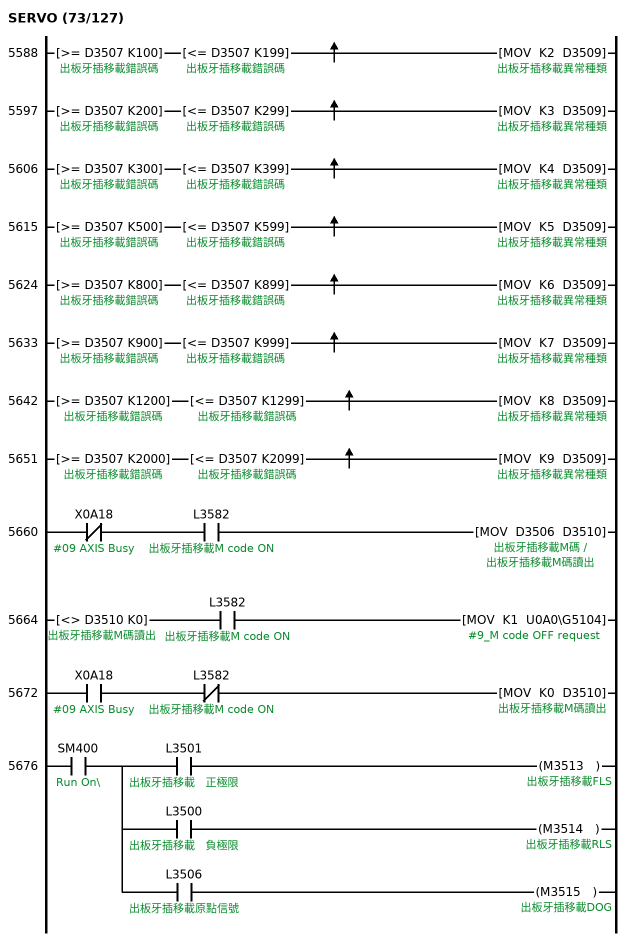
[picture p72: ladder of SERVO, rungs at steps 5588 to 5676]
5588  LD>=    D3507 K100  ; 出板牙插移載錯誤碼
      AND<=   D3507 K199  ; 出板牙插移載錯誤碼
      MEP
      MOV     K2 D3509
5597  LD>=    D3507 K200  ; 出板牙插移載錯誤碼
      AND<=   D3507 K299  ; 出板牙插移載錯誤碼
      MEP
      MOV     K3 D3509
5606  LD>=    D3507 K300  ; 出板牙插移載錯誤碼
      AND<=   D3507 K399  ; 出板牙插移載錯誤碼
      MEP
      MOV     K4 D3509
5615  LD>=    D3507 K500  ; 出板牙插移載錯誤碼
      AND<=   D3507 K599  ; 出板牙插移載錯誤碼
      MEP
      MOV     K5 D3509
5624  LD>=    D3507 K800  ; 出板牙插移載錯誤碼
      AND<=   D3507 K899  ; 出板牙插移載錯誤碼
      MEP
      MOV     K6 D3509
5633  LD>=    D3507 K900  ; 出板牙插移載錯誤碼
      AND<=   D3507 K999  ; 出板牙插移載錯誤碼
      MEP
      MOV     K7 D3509
5642  LD>=    D3507 K1200  ; 出板牙插移載錯誤碼
      AND<=   D3507 K1299  ; 出板牙插移載錯誤碼
      MEP
      MOV     K8 D3509
5651  LD>=    D3507 K2000  ; 出板牙插移載錯誤碼
      AND<=   D3507 K2099  ; 出板牙插移載錯誤碼
      MEP
      MOV     K9 D3509
5660  LDI     X0A18  ; #09 AXIS Busy
      AND     L3582  ; 出板牙插移載M code ON
      MOV     D3506 D3510  ; 出板牙插移載M碼讀出
5664  LD<>    D3510 K0  ; 出板牙插移載M碼讀出
      AND     L3582  ; 出板牙插移載M code ON
      MOV     K1 U0A0\G5104  ; #9_M code OFF request
5672  LD      X0A18  ; #09 AXIS Busy
      ANI     L3582  ; 出板牙插移載M code ON
      MOV     K0 D3510
5676  LD      SM400  ; Run On\
      MPS
      AND     L3501  ; 出板牙插移載   正極限
      OUT     M3513  ; 出板牙插移載FLS
      MRD
      AND     L3500  ; 出板牙插移載   負極限
      OUT     M3514  ; 出板牙插移載RLS
      MPP
      AND     L3506  ; 出板牙插移載原點信號
      OUT     M3515  ; 出板牙插移載DOG
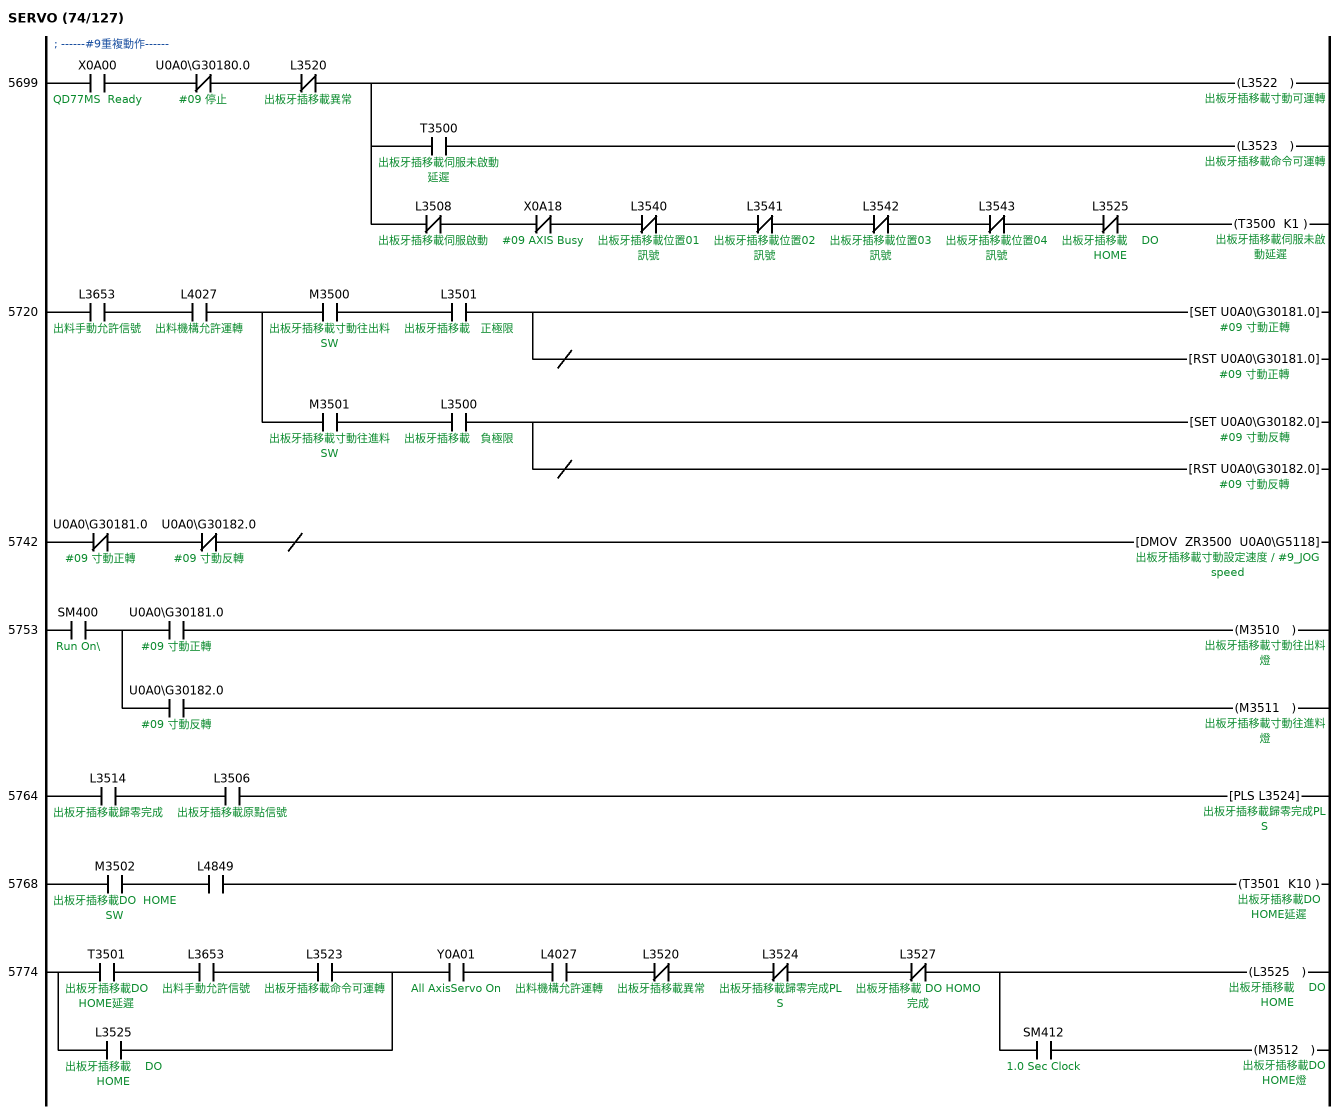
; ------#9重複動作------
5699  LD      X0A00  ; QD77MS  Ready
      ANI     U0A0\G30180.0  ; #09 停止
      ANI     L3520  ; 出板牙插移載異常
      OUT     L3522  ; 出板牙插移載寸動可運轉
      MPS
      AND     T3500  ; 出板牙插移載伺服未啟動延遲
      OUT     L3523  ; 出板牙插移載命令可運轉
      MPP
      ANI     L3508  ; 出板牙插移載伺服啟動
      ANI     X0A18  ; #09 AXIS Busy
      ANI     L3540  ; 出板牙插移載位置01 訊號
      ANI     L3541  ; 出板牙插移載位置02 訊號
      ANI     L3542  ; 出板牙插移載位置03 訊號
      ANI     L3543  ; 出板牙插移載位置04 訊號
      ANI     L3525  ; 出板牙插移載    DO HOME
      OUT     T3500 K1  ; 出板牙插移載伺服未啟動延遲
5720  LD      L3653  ; 出料手動允許信號
      AND     L4027  ; 出料機構允許運轉
      MPS
      AND     M3500  ; 出板牙插移載寸動往出料SW
      AND     L3501  ; 出板牙插移載   正極限
      SET     U0A0\G30181.0  ; #09 寸動正轉
      INV
      RST     U0A0\G30181.0  ; #09 寸動正轉
      MPP
      AND     M3501  ; 出板牙插移載寸動往進料SW
      AND     L3500  ; 出板牙插移載   負極限
      SET     U0A0\G30182.0  ; #09 寸動反轉
      INV
      RST     U0A0\G30182.0  ; #09 寸動反轉
5742  LDI     U0A0\G30181.0  ; #09 寸動正轉
      ANI     U0A0\G30182.0  ; #09 寸動反轉
      INV
      DMOV    ZR3500 U0A0\G5118  ; 出板牙插移載寸動設定速度 / #9_JOG     speed
5753  LD      SM400  ; Run On\
      MPS
      AND     U0A0\G30181.0  ; #09 寸動正轉
      OUT     M3510  ; 出板牙插移載寸動往出料燈
      MPP
      AND     U0A0\G30182.0  ; #09 寸動反轉
      OUT     M3511  ; 出板牙插移載寸動往進料燈
5764  LD      L3514  ; 出板牙插移載歸零完成
      AND     L3506  ; 出板牙插移載原點信號
      PLS     L3524  ; 出板牙插移載歸零完成PLS
5768  LD      M3502  ; 出板牙插移載DO  HOME SW
      AND     L4849
      OUT     T3501 K10  ; 出板牙插移載DO HOME延遲
5774  LD      T3501  ; 出板牙插移載DO HOME延遲
      AND     L3653  ; 出料手動允許信號
      AND     L3523  ; 出板牙插移載命令可運轉
      OR      L3525  ; 出板牙插移載    DO HOME
      AND     Y0A01  ; All AxisServo On
      AND     L4027  ; 出料機構允許運轉
      ANI     L3520  ; 出板牙插移載異常
      ANI     L3524  ; 出板牙插移載歸零完成PLS
      ANI     L3527  ; 出板牙插移載 DO HOMO 完成
      OUT     L3525  ; 出板牙插移載    DO HOME
      AND     SM412  ; 1.0 Sec Clock
      OUT     M3512  ; 出板牙插移載DO  HOME燈
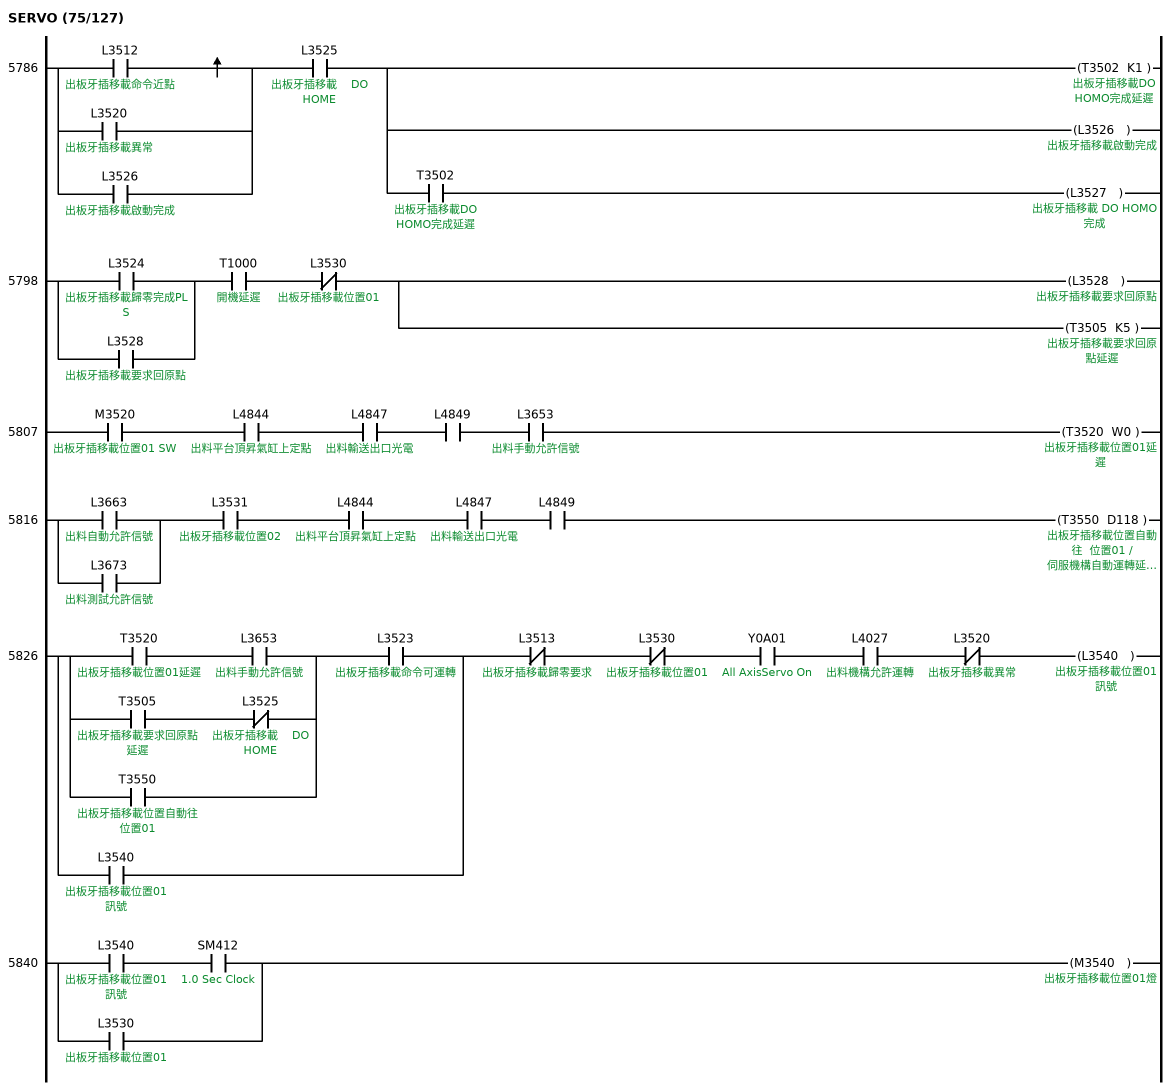
5786  LD      L3512  ; 出板牙插移載命令近點
      MEP
      OR      L3520  ; 出板牙插移載異常
      OR      L3526  ; 出板牙插移載啟動完成
      AND     L3525  ; 出板牙插移載    DO HOME
      OUT     T3502 K1  ; 出板牙插移載DO HOMO完成延遲
      OUT     L3526  ; 出板牙插移載啟動完成
      AND     T3502  ; 出板牙插移載DO HOMO完成延遲
      OUT     L3527  ; 出板牙插移載 DO HOMO 完成
5798  LD      L3524  ; 出板牙插移載歸零完成PLS
      OR      L3528  ; 出板牙插移載要求回原點
      AND     T1000  ; 開機延遲
      ANI     L3530  ; 出板牙插移載位置01
      OUT     L3528  ; 出板牙插移載要求回原點
      OUT     T3505 K5  ; 出板牙插移載要求回原點延遲
5807  LD      M3520  ; 出板牙插移載位置01 SW
      AND     L4844  ; 出料平台頂昇氣缸上定點
      AND     L4847  ; 出料輸送出口光電
      AND     L4849
      AND     L3653  ; 出料手動允許信號
      OUT     T3520 W0  ; 出板牙插移載位置01延遲
5816  LD      L3663  ; 出料自動允許信號
      OR      L3673  ; 出料測試允許信號
      AND     L3531  ; 出板牙插移載位置02
      AND     L4844  ; 出料平台頂昇氣缸上定點
      AND     L4847  ; 出料輸送出口光電
      AND     L4849
      OUT     T3550 D118  ; 出板牙插移載位置自動往  位置01 / 伺服機構自動運轉延遲時間
5826  LD      T3520  ; 出板牙插移載位置01延遲
      AND     L3653  ; 出料手動允許信號
      LD      T3505  ; 出板牙插移載要求回原點延遲
      ANI     L3525  ; 出板牙插移載    DO HOME
      ORB
      OR      T3550  ; 出板牙插移載位置自動往  位置01
      AND     L3523  ; 出板牙插移載命令可運轉
      OR      L3540  ; 出板牙插移載位置01 訊號
      ANI     L3513  ; 出板牙插移載歸零要求
      ANI     L3530  ; 出板牙插移載位置01
      AND     Y0A01  ; All AxisServo On
      AND     L4027  ; 出料機構允許運轉
      ANI     L3520  ; 出板牙插移載異常
      OUT     L3540  ; 出板牙插移載位置01 訊號
5840  LD      L3540  ; 出板牙插移載位置01 訊號
      AND     SM412  ; 1.0 Sec Clock
      OR      L3530  ; 出板牙插移載位置01
      OUT     M3540  ; 出板牙插移載位置01燈
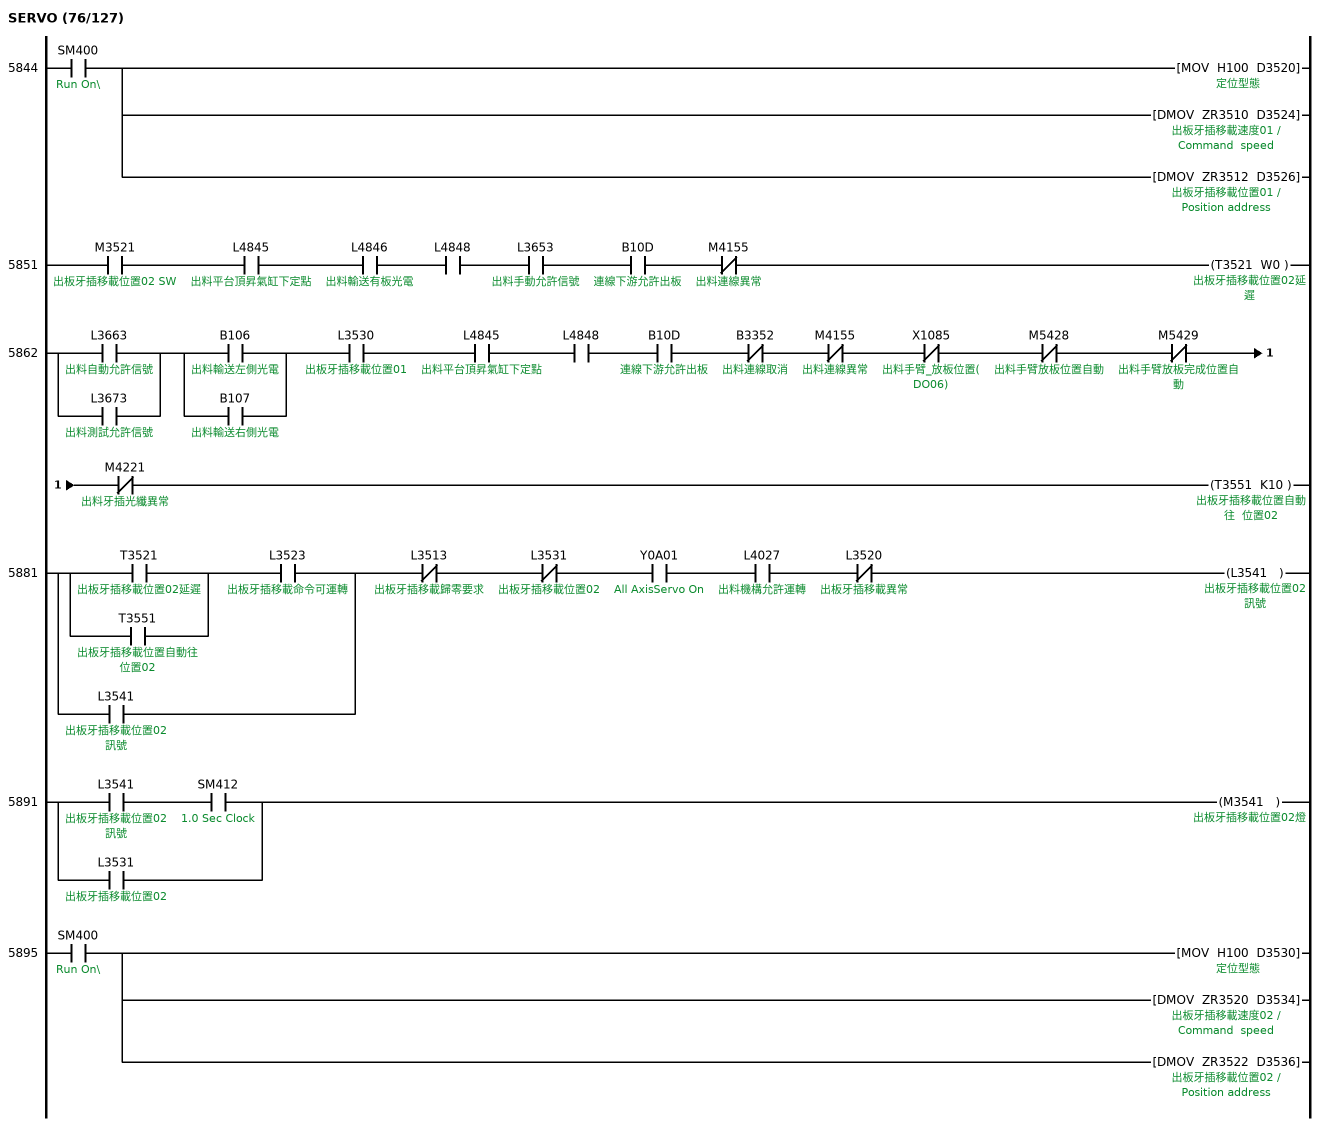
5844  LD      SM400  ; Run On\
      MOV     H100 D3520  ; 定位型態
      DMOV    ZR3510 D3524  ; 出板牙插移載速度01 / Command  speed
      DMOV    ZR3512 D3526  ; Position address
5851  LD      M3521  ; 出板牙插移載位置02 SW
      AND     L4845  ; 出料平台頂昇氣缸下定點
      AND     L4846  ; 出料輸送有板光電
      AND     L4848
      AND     L3653  ; 出料手動允許信號
      AND     B10D  ; 連線下游允許出板
      ANI     M4155  ; 出料連線異常
      OUT     T3521 W0  ; 出板牙插移載位置02延遲
5862  LD      L3663  ; 出料自動允許信號
      OR      L3673  ; 出料測試允許信號
      LD      B106  ; 出料輸送左側光電
      OR      B107  ; 出料輸送右側光電
      ANB
      AND     L3530  ; 出板牙插移載位置01
      AND     L4845  ; 出料平台頂昇氣缸下定點
      AND     L4848
      AND     B10D  ; 連線下游允許出板
      ANI     B3352  ; 出料連線取消
      ANI     M4155  ; 出料連線異常
      ANI     X1085  ; 出料手臂_放板位置(DO06)
      ANI     M5428  ; 出料手臂放板位置自動
      ANI     M5429  ; 出料手臂放板完成位置自動
      ANI     M4221  ; 出料牙插光纖異常
      OUT     T3551 K10  ; 出板牙插移載位置自動往  位置02
5881  LD      T3521  ; 出板牙插移載位置02延遲
      OR      T3551  ; 出板牙插移載位置自動往  位置02
      AND     L3523  ; 出板牙插移載命令可運轉
      OR      L3541  ; 出板牙插移載位置02 訊號
      ANI     L3513  ; 出板牙插移載歸零要求
      ANI     L3531  ; 出板牙插移載位置02
      AND     Y0A01  ; All AxisServo On
      AND     L4027  ; 出料機構允許運轉
      ANI     L3520  ; 出板牙插移載異常
      OUT     L3541  ; 出板牙插移載位置02 訊號
5891  LD      L3541  ; 出板牙插移載位置02 訊號
      AND     SM412  ; 1.0 Sec Clock
      OR      L3531  ; 出板牙插移載位置02
      OUT     M3541  ; 出板牙插移載位置02燈
5895  LD      SM400  ; Run On\
      MOV     H100 D3530  ; 定位型態
      DMOV    ZR3520 D3534  ; 出板牙插移載速度02 / Command  speed
      DMOV    ZR3522 D3536  ; Position address
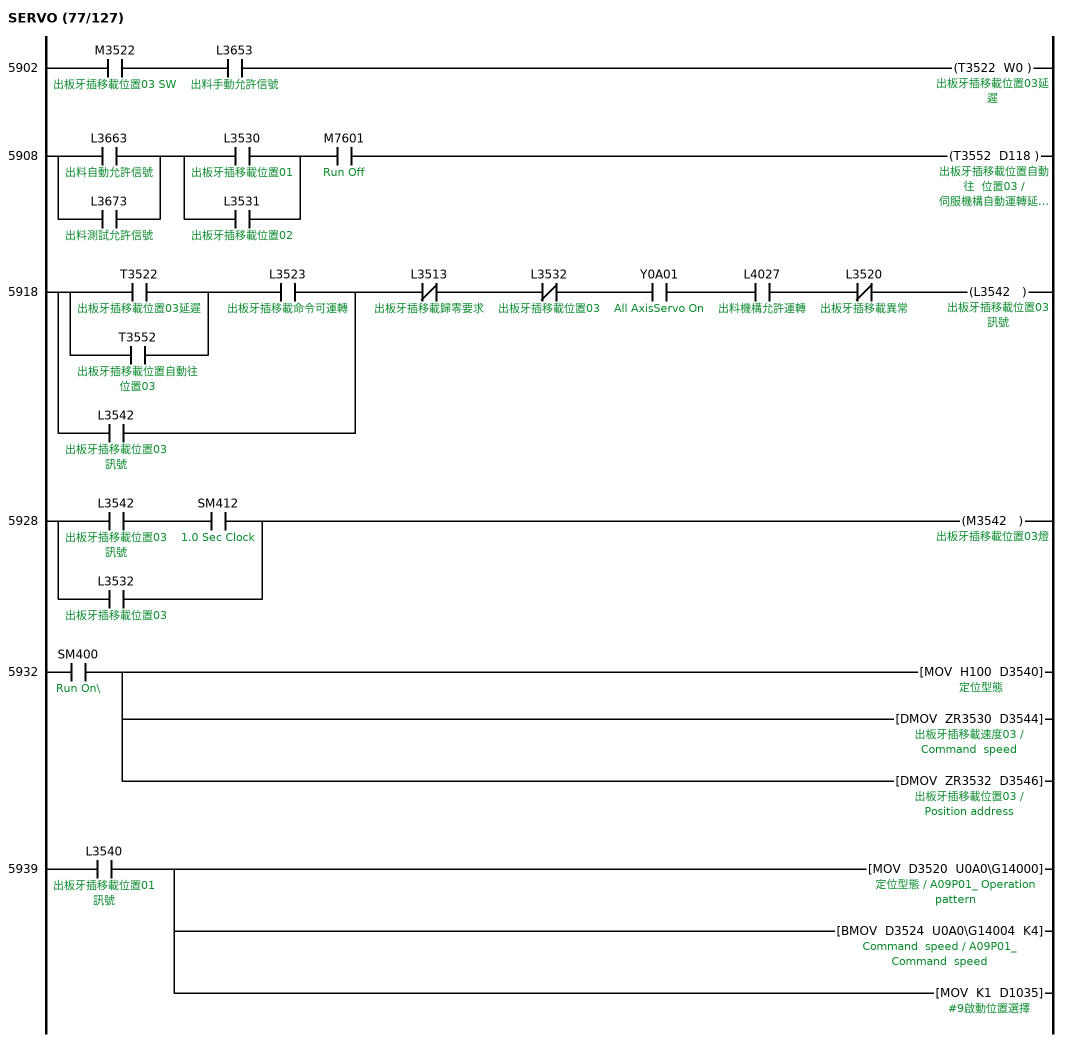
5902  LD      M3522  ; 出板牙插移載位置03 SW
      AND     L3653  ; 出料手動允許信號
      OUT     T3522 W0  ; 出板牙插移載位置03延遲
5908  LD      L3663  ; 出料自動允許信號
      OR      L3673  ; 出料測試允許信號
      LD      L3530  ; 出板牙插移載位置01
      OR      L3531  ; 出板牙插移載位置02
      ANB
      AND     M7601  ; Run Off
      OUT     T3552 D118  ; 出板牙插移載位置自動往  位置03 / 伺服機構自動運轉延遲時間
5918  LD      T3522  ; 出板牙插移載位置03延遲
      OR      T3552  ; 出板牙插移載位置自動往  位置03
      AND     L3523  ; 出板牙插移載命令可運轉
      OR      L3542  ; 出板牙插移載位置03 訊號
      ANI     L3513  ; 出板牙插移載歸零要求
      ANI     L3532  ; 出板牙插移載位置03
      AND     Y0A01  ; All AxisServo On
      AND     L4027  ; 出料機構允許運轉
      ANI     L3520  ; 出板牙插移載異常
      OUT     L3542  ; 出板牙插移載位置03 訊號
5928  LD      L3542  ; 出板牙插移載位置03 訊號
      AND     SM412  ; 1.0 Sec Clock
      OR      L3532  ; 出板牙插移載位置03
      OUT     M3542  ; 出板牙插移載位置03燈
5932  LD      SM400  ; Run On\
      MOV     H100 D3540  ; 定位型態
      DMOV    ZR3530 D3544  ; 出板牙插移載速度03 / Command  speed
      DMOV    ZR3532 D3546  ; Position address
5939  LD      L3540  ; 出板牙插移載位置01 訊號
      MOV     D3520 U0A0\G14000  ; A09P01_ Operation pattern
      BMOV    D3524 U0A0\G14004 K4  ; A09P01_ Command  speed
      MOV     K1 D1035  ; #9啟動位置選擇
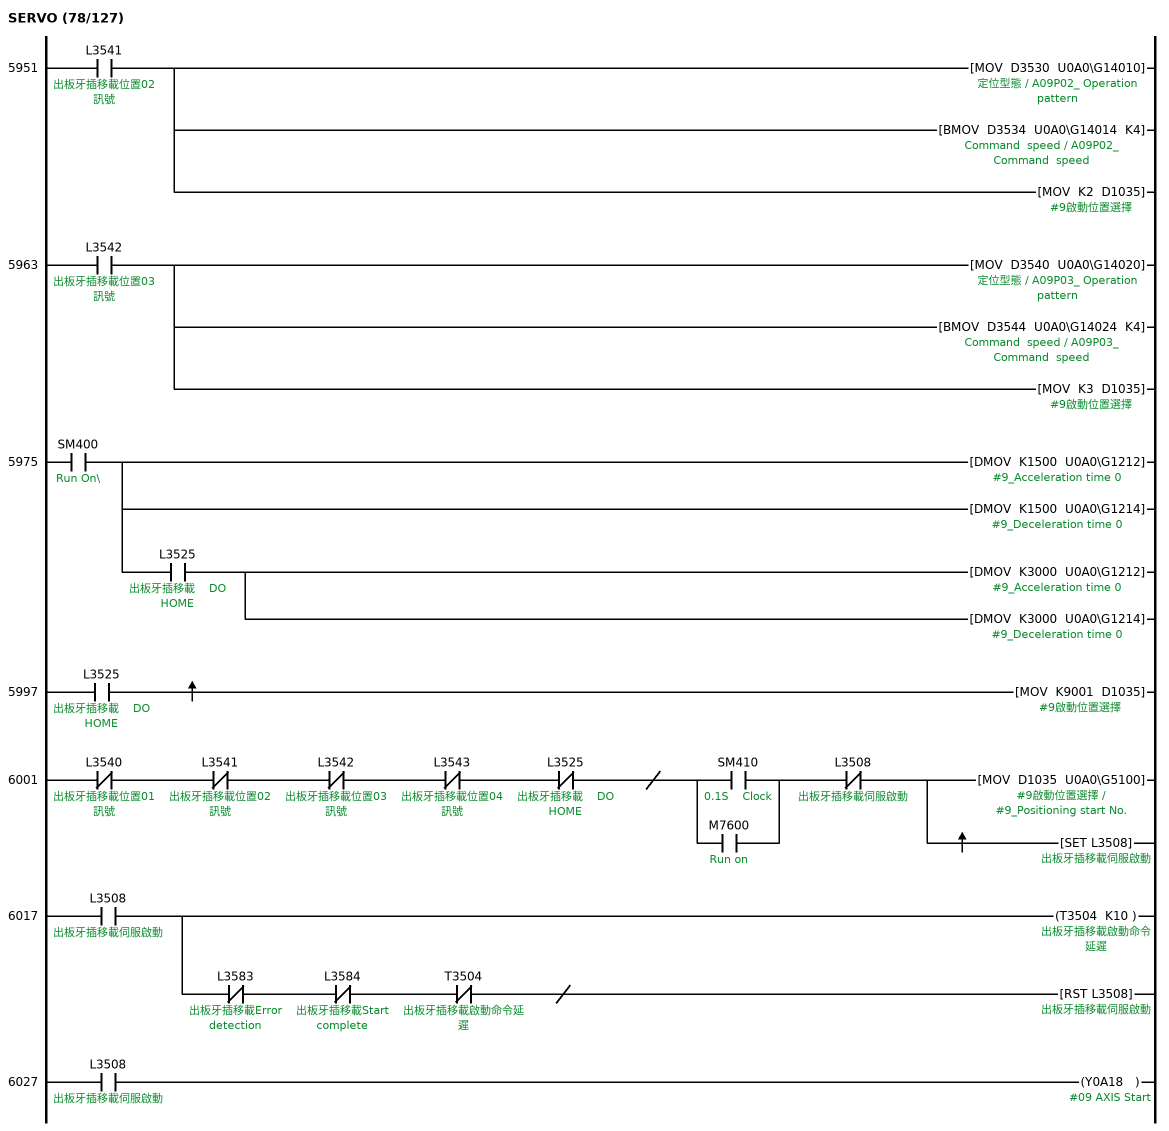
5951  LD      L3541  ; 出板牙插移載位置02 訊號
      MOV     D3530 U0A0\G14010  ; A09P02_ Operation pattern
      BMOV    D3534 U0A0\G14014 K4  ; A09P02_ Command  speed
      MOV     K2 D1035
5963  LD      L3542  ; 出板牙插移載位置03 訊號
      MOV     D3540 U0A0\G14020  ; A09P03_ Operation pattern
      BMOV    D3544 U0A0\G14024 K4  ; A09P03_ Command  speed
      MOV     K3 D1035
5975  LD      SM400  ; Run On\
      DMOV    K1500 U0A0\G1212  ; #9_Acceleration time 0
      DMOV    K1500 U0A0\G1214  ; #9_Deceleration time 0
      AND     L3525  ; 出板牙插移載    DO HOME
      DMOV    K3000 U0A0\G1212
      DMOV    K3000 U0A0\G1214
5997  LD      L3525  ; 出板牙插移載    DO HOME
      MEP
      MOV     K9001 D1035
6001  LDI     L3540  ; 出板牙插移載位置01 訊號
      ANI     L3541  ; 出板牙插移載位置02 訊號
      ANI     L3542  ; 出板牙插移載位置03 訊號
      ANI     L3543  ; 出板牙插移載位置04 訊號
      ANI     L3525  ; 出板牙插移載    DO HOME
      INV
      LD      SM410  ; 0.1S    Clock
      OR      M7600  ; Run on
      ANB
      ANI     L3508  ; 出板牙插移載伺服啟動
      MOV     D1035 U0A0\G5100  ; #9_Positioning start No.
      MEP
      SET     L3508  ; 出板牙插移載伺服啟動
6017  LD      L3508  ; 出板牙插移載伺服啟動
      OUT     T3504 K10  ; 出板牙插移載啟動命令延遲
      ANI     L3583  ; 出板牙插移載Error detection
      ANI     L3584  ; 出板牙插移載Start complete
      ANI     T3504  ; 出板牙插移載啟動命令延遲
      INV
      RST     L3508  ; 出板牙插移載伺服啟動
6027  LD      L3508  ; 出板牙插移載伺服啟動
      OUT     Y0A18  ; #09 AXIS Start
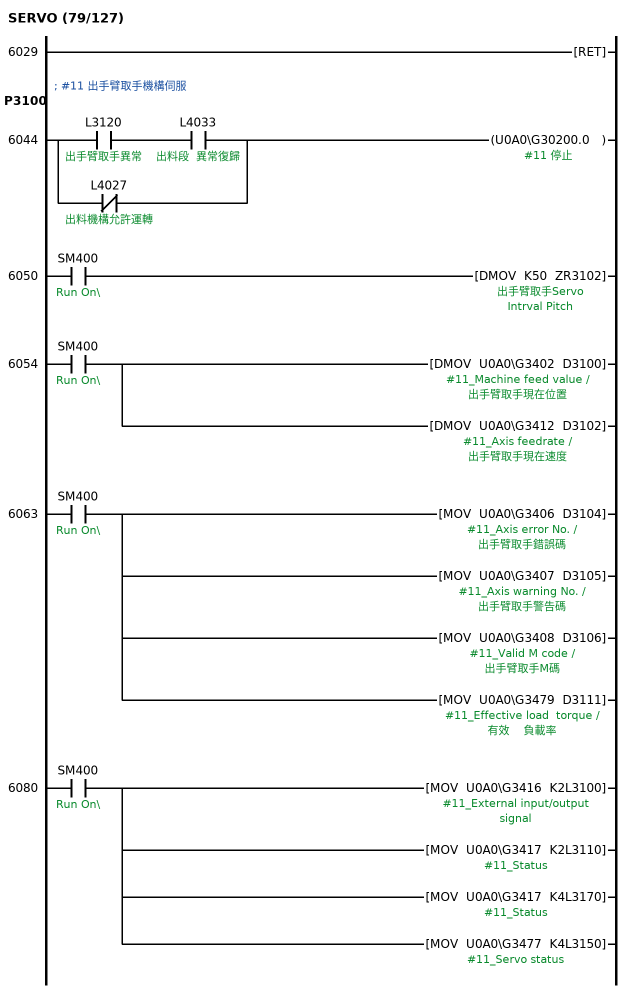
6029  RET
; #11 出手臂取手機構伺服
      P3100
6044  LD      L3120  ; 出手臂取手異常
      AND     L4033  ; 出料段  異常復歸
      ORI     L4027  ; 出料機構允許運轉
      OUT     U0A0\G30200.0  ; #11 停止
6050  LD      SM400  ; Run On\
      DMOV    K50 ZR3102  ; 出手臂取手Servo   Intrval Pitch
6054  LD      SM400  ; Run On\
      DMOV    U0A0\G3402 D3100  ; #11_Machine feed value / 出手臂取手現在位置
      DMOV    U0A0\G3412 D3102  ; #11_Axis feedrate / 出手臂取手現在速度
6063  LD      SM400  ; Run On\
      MOV     U0A0\G3406 D3104  ; #11_Axis error No. / 出手臂取手錯誤碼
      MOV     U0A0\G3407 D3105  ; #11_Axis warning No. / 出手臂取手警告碼
      MOV     U0A0\G3408 D3106  ; #11_Valid M code / 出手臂取手M碼
      MOV     U0A0\G3479 D3111  ; #11_Effective load  torque / 有效    負載率
6080  LD      SM400  ; Run On\
      MOV     U0A0\G3416 K2L3100  ; #11_External input/output signal / 出手臂取手     負極限
      MOV     U0A0\G3417 K2L3110  ; #11_Status / 出手臂取手速度控制
      MOV     U0A0\G3417 K4L3170  ; 出手臂取手速度控制
      MOV     U0A0\G3477 K4L3150  ; #11_Servo status / READY ON
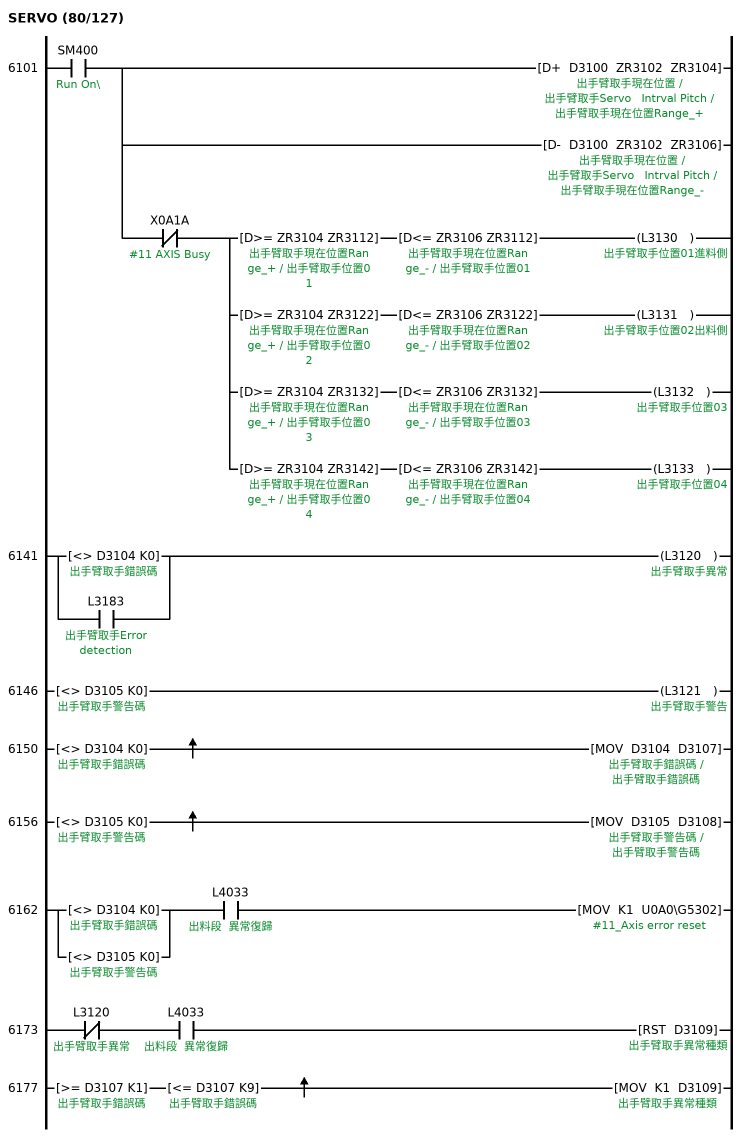
6101  LD      SM400  ; Run On\
      D+      D3100 ZR3102 ZR3104  ; 出手臂取手現在位置Range_+
      D-      D3100 ZR3102 ZR3106  ; 出手臂取手現在位置Range_-
      ANI     X0A1A  ; #11 AXIS Busy
      MPS
      ANDD>=  ZR3104 ZR3112  ; 出手臂取手現在位置Range_+ / 出手臂取手位置01
      ANDD<=  ZR3106 ZR3112  ; 出手臂取手現在位置Range_- / 出手臂取手位置01
      OUT     L3130  ; 出手臂取手位置01進料側
      MRD
      ANDD>=  ZR3104 ZR3122  ; 出手臂取手現在位置Range_+ / 出手臂取手位置02
      ANDD<=  ZR3106 ZR3122  ; 出手臂取手現在位置Range_- / 出手臂取手位置02
      OUT     L3131  ; 出手臂取手位置02出料側
      MRD
      ANDD>=  ZR3104 ZR3132  ; 出手臂取手現在位置Range_+ / 出手臂取手位置03
      ANDD<=  ZR3106 ZR3132  ; 出手臂取手現在位置Range_- / 出手臂取手位置03
      OUT     L3132  ; 出手臂取手位置03
      MPP
      ANDD>=  ZR3104 ZR3142  ; 出手臂取手現在位置Range_+ / 出手臂取手位置04
      ANDD<=  ZR3106 ZR3142  ; 出手臂取手現在位置Range_- / 出手臂取手位置04
      OUT     L3133  ; 出手臂取手位置04
6141  LD<>    D3104 K0  ; 出手臂取手錯誤碼
      OR      L3183  ; 出手臂取手Error detection
      OUT     L3120  ; 出手臂取手異常
6146  LD<>    D3105 K0  ; 出手臂取手警告碼
      OUT     L3121  ; 出手臂取手警告
6150  LD<>    D3104 K0  ; 出手臂取手錯誤碼
      MEP
      MOV     D3104 D3107  ; 出手臂取手錯誤碼
6156  LD<>    D3105 K0  ; 出手臂取手警告碼
      MEP
      MOV     D3105 D3108  ; 出手臂取手警告碼
6162  LD<>    D3104 K0  ; 出手臂取手錯誤碼
      OR<>    D3105 K0  ; 出手臂取手警告碼
      AND     L4033  ; 出料段  異常復歸
      MOV     K1 U0A0\G5302  ; #11_Axis error reset
6173  LDI     L3120  ; 出手臂取手異常
      AND     L4033  ; 出料段  異常復歸
      RST     D3109  ; 出手臂取手異常種類
6177  LD>=    D3107 K1  ; 出手臂取手錯誤碼
      AND<=   D3107 K9  ; 出手臂取手錯誤碼
      MEP
      MOV     K1 D3109
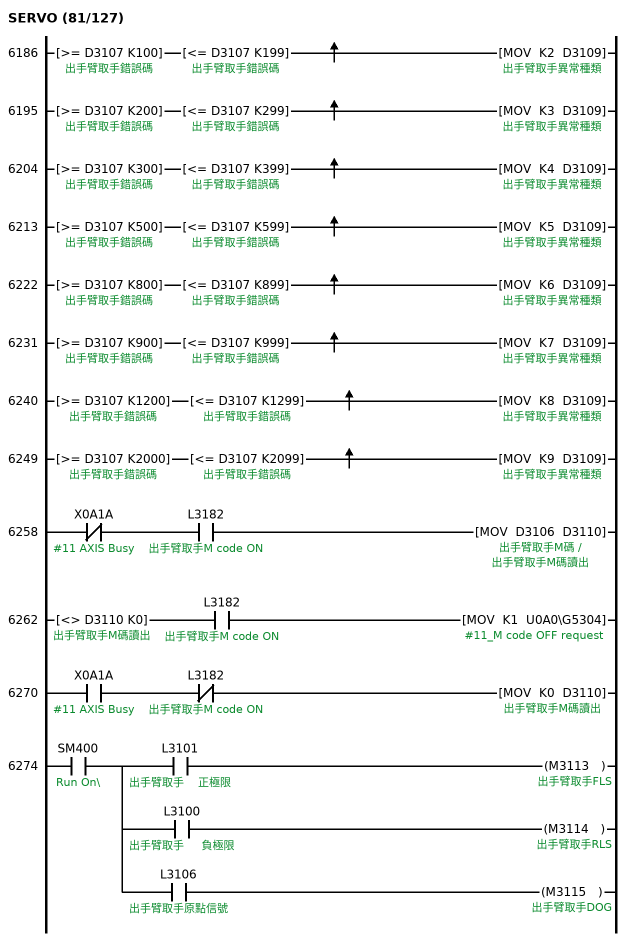
6186  LD>=    D3107 K100  ; 出手臂取手錯誤碼
      AND<=   D3107 K199  ; 出手臂取手錯誤碼
      MEP
      MOV     K2 D3109
6195  LD>=    D3107 K200  ; 出手臂取手錯誤碼
      AND<=   D3107 K299  ; 出手臂取手錯誤碼
      MEP
      MOV     K3 D3109
6204  LD>=    D3107 K300  ; 出手臂取手錯誤碼
      AND<=   D3107 K399  ; 出手臂取手錯誤碼
      MEP
      MOV     K4 D3109
6213  LD>=    D3107 K500  ; 出手臂取手錯誤碼
      AND<=   D3107 K599  ; 出手臂取手錯誤碼
      MEP
      MOV     K5 D3109
6222  LD>=    D3107 K800  ; 出手臂取手錯誤碼
      AND<=   D3107 K899  ; 出手臂取手錯誤碼
      MEP
      MOV     K6 D3109
6231  LD>=    D3107 K900  ; 出手臂取手錯誤碼
      AND<=   D3107 K999  ; 出手臂取手錯誤碼
      MEP
      MOV     K7 D3109
6240  LD>=    D3107 K1200  ; 出手臂取手錯誤碼
      AND<=   D3107 K1299  ; 出手臂取手錯誤碼
      MEP
      MOV     K8 D3109
6249  LD>=    D3107 K2000  ; 出手臂取手錯誤碼
      AND<=   D3107 K2099  ; 出手臂取手錯誤碼
      MEP
      MOV     K9 D3109
6258  LDI     X0A1A  ; #11 AXIS Busy
      AND     L3182  ; 出手臂取手M code ON
      MOV     D3106 D3110  ; 出手臂取手M碼讀出
6262  LD<>    D3110 K0  ; 出手臂取手M碼讀出
      AND     L3182  ; 出手臂取手M code ON
      MOV     K1 U0A0\G5304  ; #11_M code OFF request
6270  LD      X0A1A  ; #11 AXIS Busy
      ANI     L3182  ; 出手臂取手M code ON
      MOV     K0 D3110
6274  LD      SM400  ; Run On\
      MPS
      AND     L3101  ; 出手臂取手    正極限
      OUT     M3113  ; 出手臂取手FLS
      MRD
      AND     L3100  ; 出手臂取手     負極限
      OUT     M3114  ; 出手臂取手RLS
      MPP
      AND     L3106  ; 出手臂取手原點信號
      OUT     M3115  ; 出手臂取手DOG
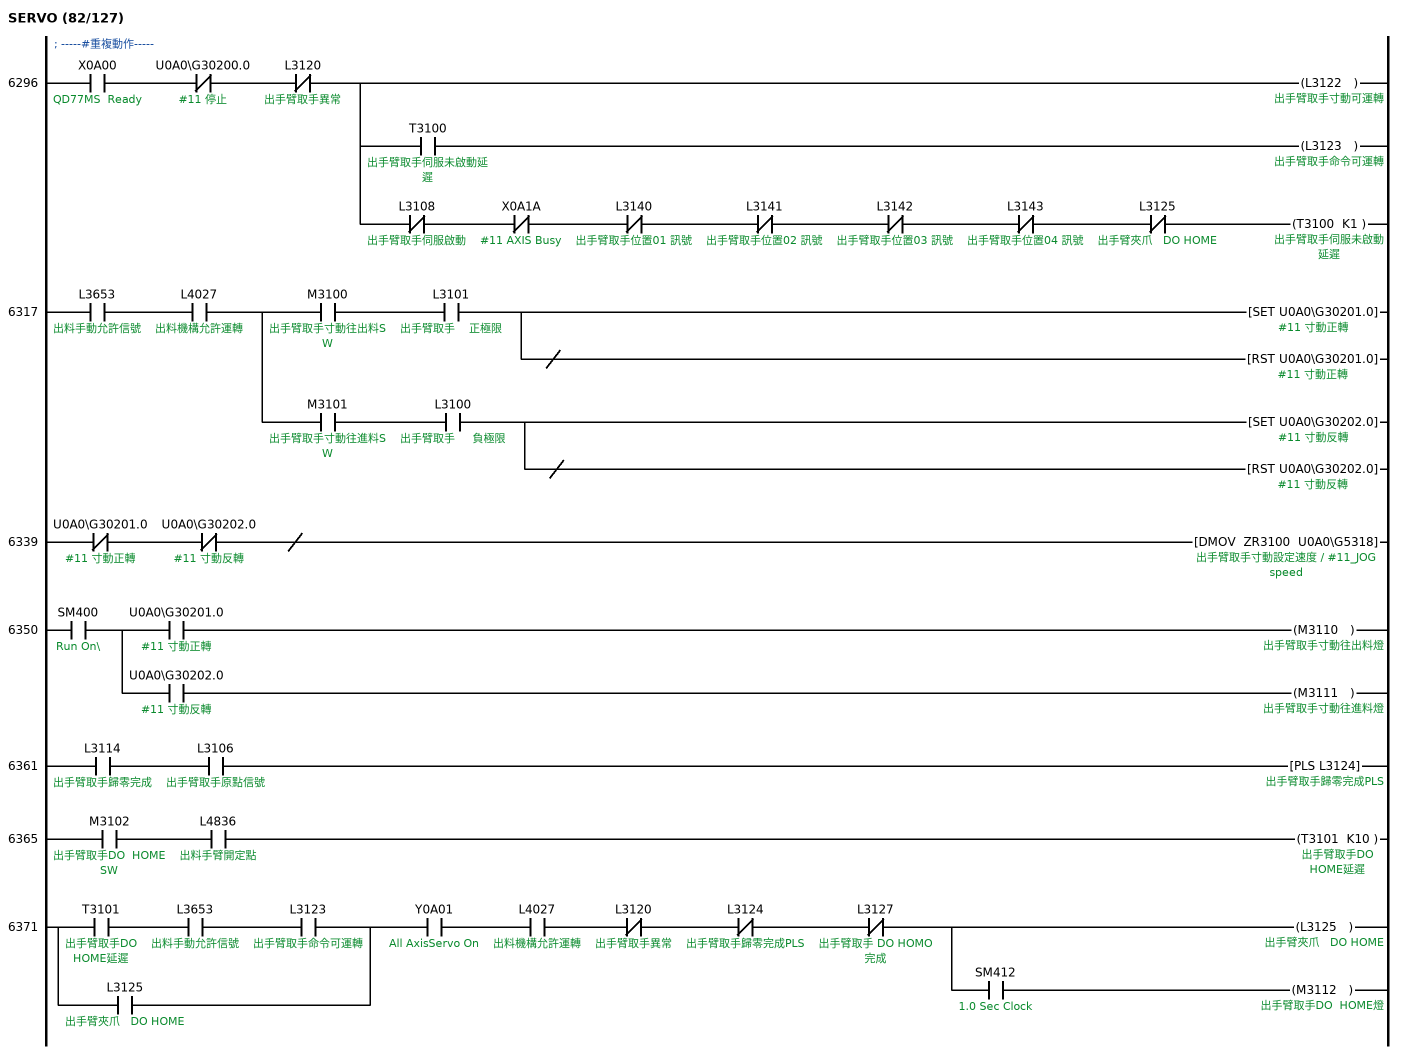
; -----#重複動作-----
6296  LD      X0A00  ; QD77MS  Ready
      ANI     U0A0\G30200.0  ; #11 停止
      ANI     L3120  ; 出手臂取手異常
      OUT     L3122  ; 出手臂取手寸動可運轉
      MPS
      AND     T3100  ; 出手臂取手伺服未啟動延遲
      OUT     L3123  ; 出手臂取手命令可運轉
      MPP
      ANI     L3108  ; 出手臂取手伺服啟動
      ANI     X0A1A  ; #11 AXIS Busy
      ANI     L3140  ; 出手臂取手位置01 訊號
      ANI     L3141  ; 出手臂取手位置02 訊號
      ANI     L3142  ; 出手臂取手位置03 訊號
      ANI     L3143  ; 出手臂取手位置04 訊號
      ANI     L3125  ; 出手臂夾爪   DO HOME
      OUT     T3100 K1  ; 出手臂取手伺服未啟動延遲
6317  LD      L3653  ; 出料手動允許信號
      AND     L4027  ; 出料機構允許運轉
      MPS
      AND     M3100  ; 出手臂取手寸動往出料SW
      AND     L3101  ; 出手臂取手    正極限
      SET     U0A0\G30201.0  ; #11 寸動正轉
      INV
      RST     U0A0\G30201.0  ; #11 寸動正轉
      MPP
      AND     M3101  ; 出手臂取手寸動往進料SW
      AND     L3100  ; 出手臂取手     負極限
      SET     U0A0\G30202.0  ; #11 寸動反轉
      INV
      RST     U0A0\G30202.0  ; #11 寸動反轉
6339  LDI     U0A0\G30201.0  ; #11 寸動正轉
      ANI     U0A0\G30202.0  ; #11 寸動反轉
      INV
      DMOV    ZR3100 U0A0\G5318  ; 出手臂取手寸動設定速度 / #11_JOG     speed
6350  LD      SM400  ; Run On\
      MPS
      AND     U0A0\G30201.0  ; #11 寸動正轉
      OUT     M3110  ; 出手臂取手寸動往出料燈
      MPP
      AND     U0A0\G30202.0  ; #11 寸動反轉
      OUT     M3111  ; 出手臂取手寸動往進料燈
6361  LD      L3114  ; 出手臂取手歸零完成
      AND     L3106  ; 出手臂取手原點信號
      PLS     L3124  ; 出手臂取手歸零完成PLS
6365  LD      M3102  ; 出手臂取手DO  HOME SW
      AND     L4836  ; 出料手臂開定點
      OUT     T3101 K10  ; 出手臂取手DO HOME延遲
6371  LD      T3101  ; 出手臂取手DO HOME延遲
      AND     L3653  ; 出料手動允許信號
      AND     L3123  ; 出手臂取手命令可運轉
      OR      L3125  ; 出手臂夾爪   DO HOME
      AND     Y0A01  ; All AxisServo On
      AND     L4027  ; 出料機構允許運轉
      ANI     L3120  ; 出手臂取手異常
      ANI     L3124  ; 出手臂取手歸零完成PLS
      ANI     L3127  ; 出手臂取手 DO HOMO 完成
      OUT     L3125  ; 出手臂夾爪   DO HOME
      AND     SM412  ; 1.0 Sec Clock
      OUT     M3112  ; 出手臂取手DO  HOME燈
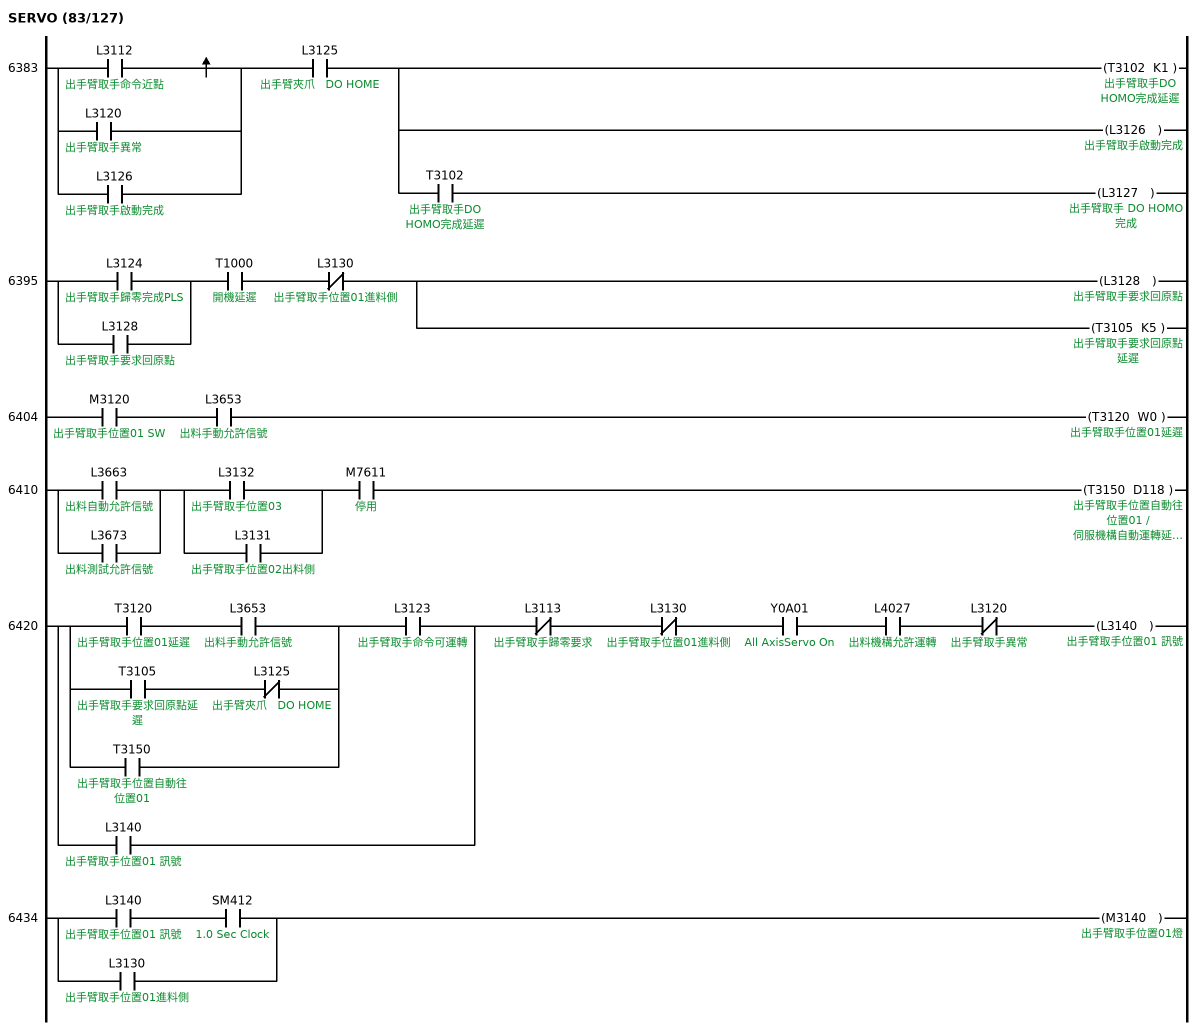
6383  LD      L3112  ; 出手臂取手命令近點
      MEP
      OR      L3120  ; 出手臂取手異常
      OR      L3126  ; 出手臂取手啟動完成
      AND     L3125  ; 出手臂夾爪   DO HOME
      OUT     T3102 K1  ; 出手臂取手DO HOMO完成延遲
      OUT     L3126  ; 出手臂取手啟動完成
      AND     T3102  ; 出手臂取手DO HOMO完成延遲
      OUT     L3127  ; 出手臂取手 DO HOMO 完成
6395  LD      L3124  ; 出手臂取手歸零完成PLS
      OR      L3128  ; 出手臂取手要求回原點
      AND     T1000  ; 開機延遲
      ANI     L3130  ; 出手臂取手位置01進料側
      OUT     L3128  ; 出手臂取手要求回原點
      OUT     T3105 K5  ; 出手臂取手要求回原點延遲
6404  LD      M3120  ; 出手臂取手位置01 SW
      AND     L3653  ; 出料手動允許信號
      OUT     T3120 W0  ; 出手臂取手位置01延遲
6410  LD      L3663  ; 出料自動允許信號
      OR      L3673  ; 出料測試允許信號
      LD      L3132  ; 出手臂取手位置03
      OR      L3131  ; 出手臂取手位置02出料側
      ANB
      AND     M7611  ; 停用
      OUT     T3150 D118  ; 出手臂取手位置自動往  位置01 / 伺服機構自動運轉延遲時間
6420  LD      T3120  ; 出手臂取手位置01延遲
      AND     L3653  ; 出料手動允許信號
      LD      T3105  ; 出手臂取手要求回原點延遲
      ANI     L3125  ; 出手臂夾爪   DO HOME
      ORB
      OR      T3150  ; 出手臂取手位置自動往  位置01
      AND     L3123  ; 出手臂取手命令可運轉
      OR      L3140  ; 出手臂取手位置01 訊號
      ANI     L3113  ; 出手臂取手歸零要求
      ANI     L3130  ; 出手臂取手位置01進料側
      AND     Y0A01  ; All AxisServo On
      AND     L4027  ; 出料機構允許運轉
      ANI     L3120  ; 出手臂取手異常
      OUT     L3140  ; 出手臂取手位置01 訊號
6434  LD      L3140  ; 出手臂取手位置01 訊號
      AND     SM412  ; 1.0 Sec Clock
      OR      L3130  ; 出手臂取手位置01進料側
      OUT     M3140  ; 出手臂取手位置01燈
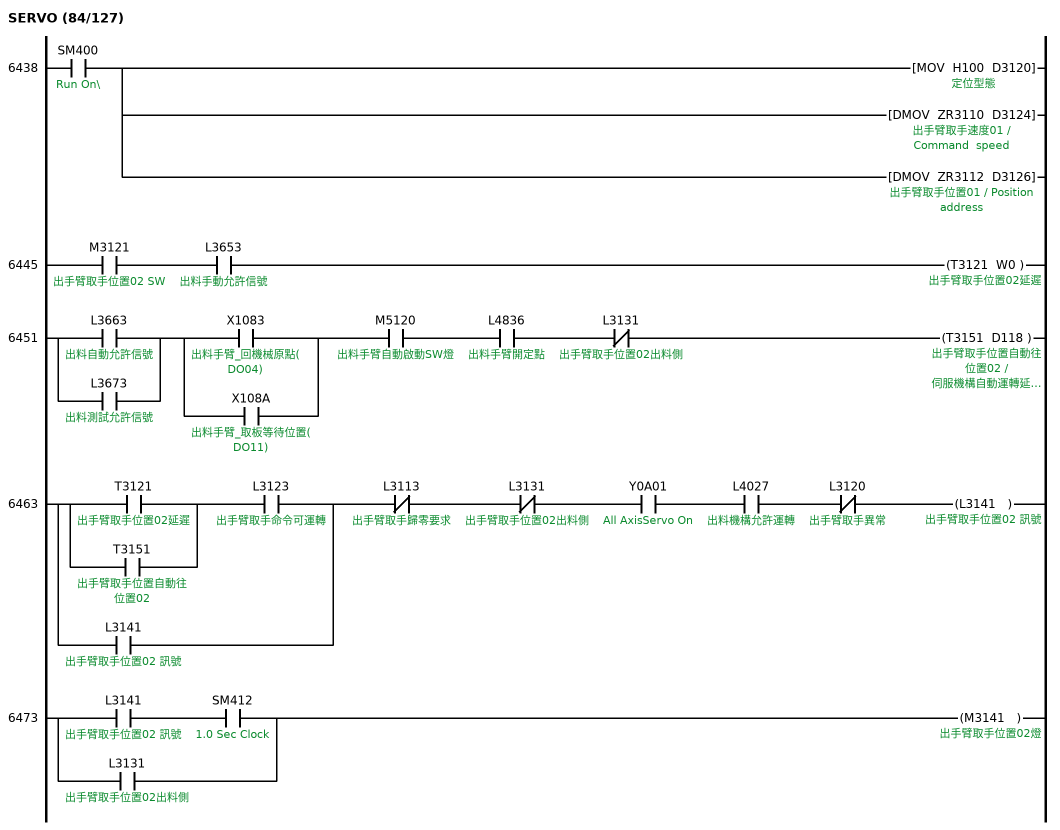
6438  LD      SM400  ; Run On\
      MOV     H100 D3120  ; 定位型態
      DMOV    ZR3110 D3124  ; 出手臂取手速度01 / Command  speed
      DMOV    ZR3112 D3126  ; Position address
6445  LD      M3121  ; 出手臂取手位置02 SW
      AND     L3653  ; 出料手動允許信號
      OUT     T3121 W0  ; 出手臂取手位置02延遲
6451  LD      L3663  ; 出料自動允許信號
      OR      L3673  ; 出料測試允許信號
      LD      X1083  ; 出料手臂_回機械原點(DO04)
      OR      X108A  ; 出料手臂_取板等待位置(DO11)
      ANB
      AND     M5120  ; 出料手臂自動啟動SW燈
      AND     L4836  ; 出料手臂開定點
      ANI     L3131  ; 出手臂取手位置02出料側
      OUT     T3151 D118  ; 出手臂取手位置自動往  位置02 / 伺服機構自動運轉延遲時間
6463  LD      T3121  ; 出手臂取手位置02延遲
      OR      T3151  ; 出手臂取手位置自動往  位置02
      AND     L3123  ; 出手臂取手命令可運轉
      OR      L3141  ; 出手臂取手位置02 訊號
      ANI     L3113  ; 出手臂取手歸零要求
      ANI     L3131  ; 出手臂取手位置02出料側
      AND     Y0A01  ; All AxisServo On
      AND     L4027  ; 出料機構允許運轉
      ANI     L3120  ; 出手臂取手異常
      OUT     L3141  ; 出手臂取手位置02 訊號
6473  LD      L3141  ; 出手臂取手位置02 訊號
      AND     SM412  ; 1.0 Sec Clock
      OR      L3131  ; 出手臂取手位置02出料側
      OUT     M3141  ; 出手臂取手位置02燈
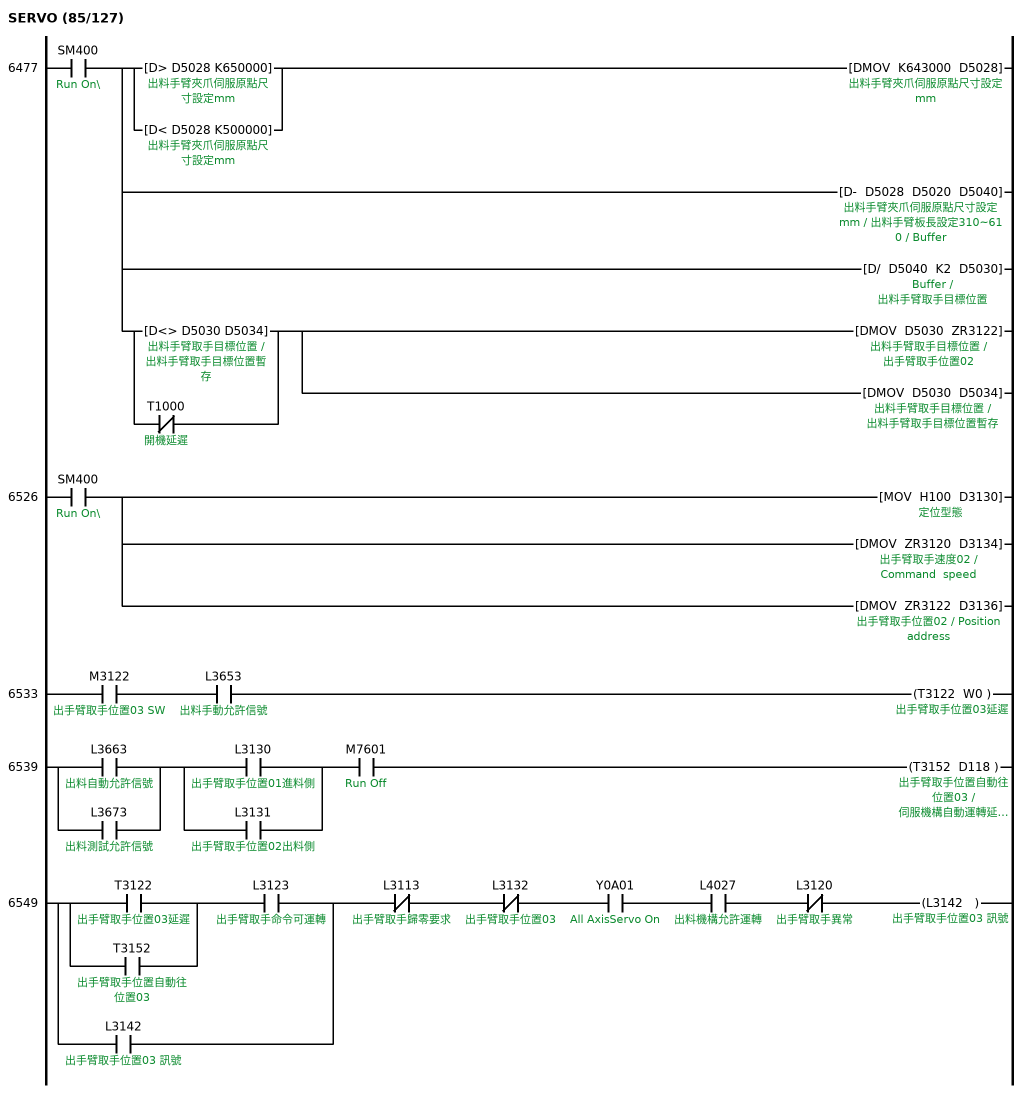
6477  LD      SM400  ; Run On\
      MPS
      LDD>    D5028 K650000  ; 出料手臂夾爪伺服原點尺寸設定mm
      ORD<    D5028 K500000  ; 出料手臂夾爪伺服原點尺寸設定mm
      ANB
      DMOV    K643000 D5028
        [note] /* 手臂夾爪伺服原點尺寸_643mm */
      MPP
      D-      D5028 D5020 D5040  ; 出料手臂板長設定310~610
      D/      D5040 K2 D5030  ; 出料手臂取手目標位置
      LDD<>   D5030 D5034  ; 出料手臂取手目標位置 / 出料手臂取手目標位置暫存
      ORI     T1000  ; 開機延遲
      ANB
      DMOV    D5030 ZR3122
      DMOV    D5030 D5034
6526  LD      SM400  ; Run On\
      MOV     H100 D3130  ; 定位型態
      DMOV    ZR3120 D3134  ; 出手臂取手速度02 / Command  speed
      DMOV    ZR3122 D3136  ; Position address
6533  LD      M3122  ; 出手臂取手位置03 SW
      AND     L3653  ; 出料手動允許信號
      OUT     T3122 W0  ; 出手臂取手位置03延遲
6539  LD      L3663  ; 出料自動允許信號
      OR      L3673  ; 出料測試允許信號
      LD      L3130  ; 出手臂取手位置01進料側
      OR      L3131  ; 出手臂取手位置02出料側
      ANB
      AND     M7601  ; Run Off
      OUT     T3152 D118  ; 出手臂取手位置自動往  位置03 / 伺服機構自動運轉延遲時間
6549  LD      T3122  ; 出手臂取手位置03延遲
      OR      T3152  ; 出手臂取手位置自動往  位置03
      AND     L3123  ; 出手臂取手命令可運轉
      OR      L3142  ; 出手臂取手位置03 訊號
      ANI     L3113  ; 出手臂取手歸零要求
      ANI     L3132  ; 出手臂取手位置03
      AND     Y0A01  ; All AxisServo On
      AND     L4027  ; 出料機構允許運轉
      ANI     L3120  ; 出手臂取手異常
      OUT     L3142  ; 出手臂取手位置03 訊號
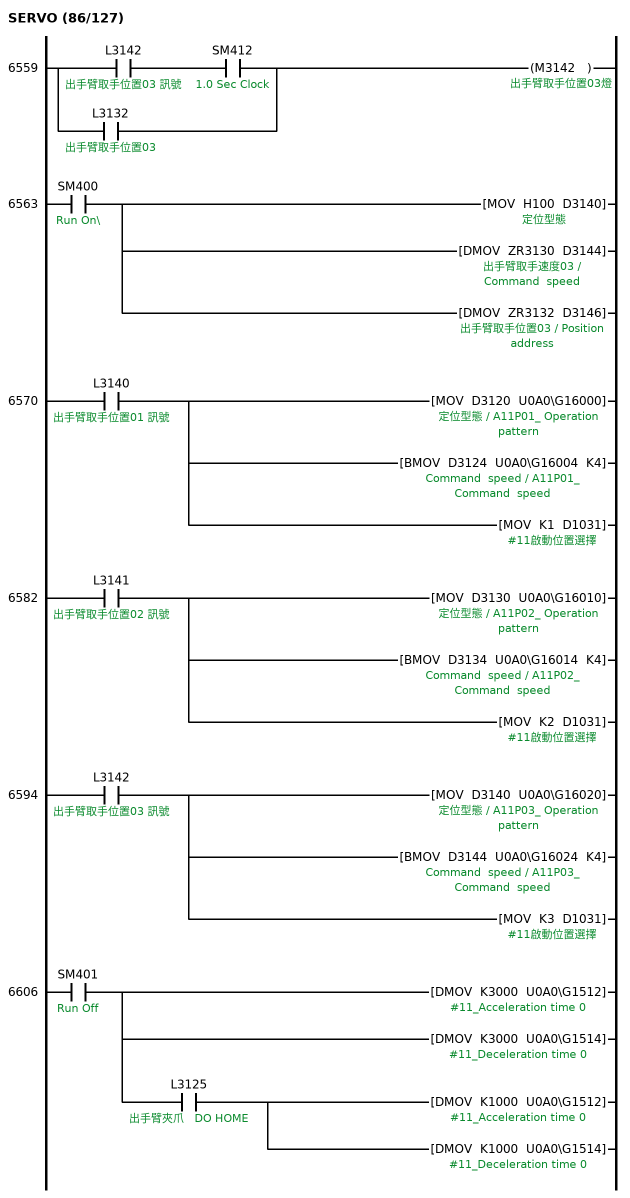
6559  LD      L3142  ; 出手臂取手位置03 訊號
      AND     SM412  ; 1.0 Sec Clock
      OR      L3132  ; 出手臂取手位置03
      OUT     M3142  ; 出手臂取手位置03燈
6563  LD      SM400  ; Run On\
      MOV     H100 D3140  ; 定位型態
      DMOV    ZR3130 D3144  ; 出手臂取手速度03 / Command  speed
      DMOV    ZR3132 D3146  ; Position address
6570  LD      L3140  ; 出手臂取手位置01 訊號
      MOV     D3120 U0A0\G16000  ; A11P01_ Operation pattern
      BMOV    D3124 U0A0\G16004 K4  ; A11P01_ Command  speed
      MOV     K1 D1031  ; #11啟動位置選擇
6582  LD      L3141  ; 出手臂取手位置02 訊號
      MOV     D3130 U0A0\G16010  ; A11P02_ Operation pattern
      BMOV    D3134 U0A0\G16014 K4  ; A11P02_ Command  speed
      MOV     K2 D1031
6594  LD      L3142  ; 出手臂取手位置03 訊號
      MOV     D3140 U0A0\G16020  ; A11P03_ Operation pattern
      BMOV    D3144 U0A0\G16024 K4  ; A11P03_ Command  speed
      MOV     K3 D1031
6606  LD      SM401  ; Run Off
      DMOV    K3000 U0A0\G1512  ; #11_Acceleration time 0
      DMOV    K3000 U0A0\G1514  ; #11_Deceleration time 0
      AND     L3125  ; 出手臂夾爪   DO HOME
      DMOV    K1000 U0A0\G1512
      DMOV    K1000 U0A0\G1514
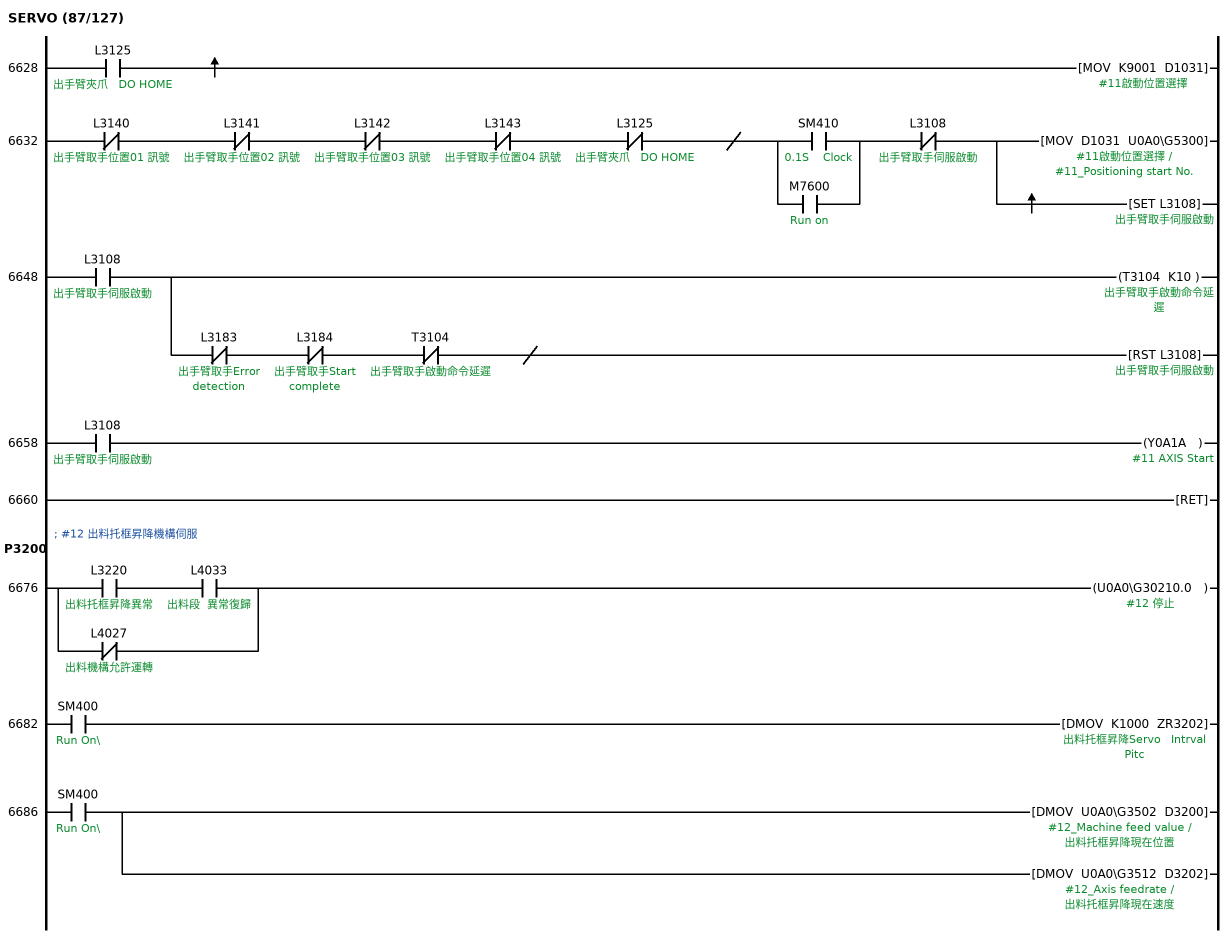
6628  LD      L3125  ; 出手臂夾爪   DO HOME
      MEP
      MOV     K9001 D1031
6632  LDI     L3140  ; 出手臂取手位置01 訊號
      ANI     L3141  ; 出手臂取手位置02 訊號
      ANI     L3142  ; 出手臂取手位置03 訊號
      ANI     L3143  ; 出手臂取手位置04 訊號
      ANI     L3125  ; 出手臂夾爪   DO HOME
      INV
      LD      SM410  ; 0.1S    Clock
      OR      M7600  ; Run on
      ANB
      ANI     L3108  ; 出手臂取手伺服啟動
      MOV     D1031 U0A0\G5300  ; #11_Positioning start No.
      MEP
      SET     L3108  ; 出手臂取手伺服啟動
6648  LD      L3108  ; 出手臂取手伺服啟動
      OUT     T3104 K10  ; 出手臂取手啟動命令延遲
      ANI     L3183  ; 出手臂取手Error detection
      ANI     L3184  ; 出手臂取手Start complete
      ANI     T3104  ; 出手臂取手啟動命令延遲
      INV
      RST     L3108  ; 出手臂取手伺服啟動
6658  LD      L3108  ; 出手臂取手伺服啟動
      OUT     Y0A1A  ; #11 AXIS Start
6660  RET
; #12 出料托框昇降機構伺服
      P3200
6676  LD      L3220  ; 出料托框昇降異常
      AND     L4033  ; 出料段  異常復歸
      ORI     L4027  ; 出料機構允許運轉
      OUT     U0A0\G30210.0  ; #12 停止
6682  LD      SM400  ; Run On\
      DMOV    K1000 ZR3202  ; 出料托框昇降Servo   Intrval Pitc
6686  LD      SM400  ; Run On\
      DMOV    U0A0\G3502 D3200  ; #12_Machine feed value / 出料托框昇降現在位置
      DMOV    U0A0\G3512 D3202  ; #12_Axis feedrate / 出料托框昇降現在速度
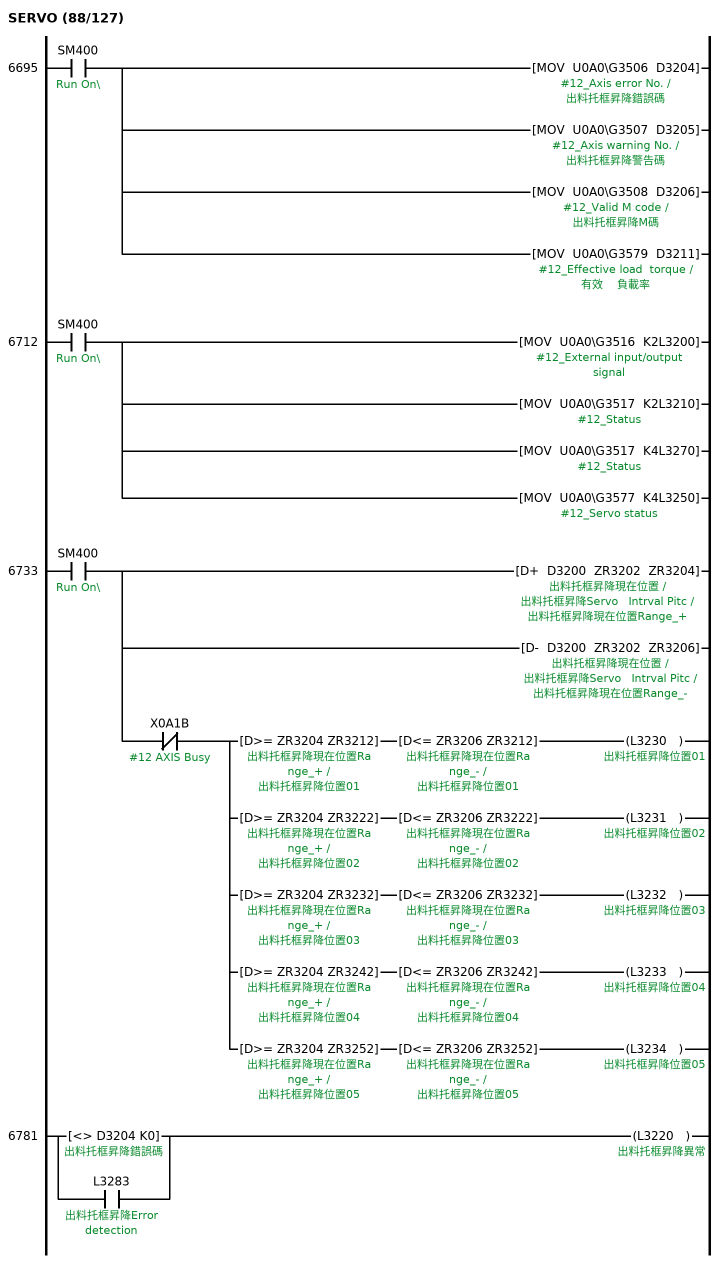
6695  LD      SM400  ; Run On\
      MOV     U0A0\G3506 D3204  ; #12_Axis error No. / 出料托框昇降錯誤碼
      MOV     U0A0\G3507 D3205  ; #12_Axis warning No. / 出料托框昇降警告碼
      MOV     U0A0\G3508 D3206  ; #12_Valid M code / 出料托框昇降M碼
      MOV     U0A0\G3579 D3211  ; #12_Effective load  torque / 有效    負載率
6712  LD      SM400  ; Run On\
      MOV     U0A0\G3516 K2L3200  ; #12_External input/output signal / 出料托框昇降    負極限
      MOV     U0A0\G3517 K2L3210  ; #12_Status / 出料托框昇降速度控制
      MOV     U0A0\G3517 K4L3270  ; 出料托框昇降速度控制
      MOV     U0A0\G3577 K4L3250  ; #12_Servo status / READY ON
6733  LD      SM400  ; Run On\
      D+      D3200 ZR3202 ZR3204  ; 出料托框昇降現在位置Range_+
      D-      D3200 ZR3202 ZR3206  ; 出料托框昇降現在位置Range_-
      ANI     X0A1B  ; #12 AXIS Busy
      MPS
      ANDD>=  ZR3204 ZR3212  ; 出料托框昇降現在位置Range_+ / 出料托框昇降位置01
      ANDD<=  ZR3206 ZR3212  ; 出料托框昇降現在位置Range_- / 出料托框昇降位置01
      OUT     L3230  ; 出料托框昇降位置01
      MRD
      ANDD>=  ZR3204 ZR3222  ; 出料托框昇降現在位置Range_+ / 出料托框昇降位置02
      ANDD<=  ZR3206 ZR3222  ; 出料托框昇降現在位置Range_- / 出料托框昇降位置02
      OUT     L3231  ; 出料托框昇降位置02
      MRD
      ANDD>=  ZR3204 ZR3232  ; 出料托框昇降現在位置Range_+ / 出料托框昇降位置03
      ANDD<=  ZR3206 ZR3232  ; 出料托框昇降現在位置Range_- / 出料托框昇降位置03
      OUT     L3232  ; 出料托框昇降位置03
      MRD
      ANDD>=  ZR3204 ZR3242  ; 出料托框昇降現在位置Range_+ / 出料托框昇降位置04
      ANDD<=  ZR3206 ZR3242  ; 出料托框昇降現在位置Range_- / 出料托框昇降位置04
      OUT     L3233  ; 出料托框昇降位置04
      MPP
      ANDD>=  ZR3204 ZR3252  ; 出料托框昇降現在位置Range_+ / 出料托框昇降位置05
      ANDD<=  ZR3206 ZR3252  ; 出料托框昇降現在位置Range_- / 出料托框昇降位置05
      OUT     L3234  ; 出料托框昇降位置05
6781  LD<>    D3204 K0  ; 出料托框昇降錯誤碼
      OR      L3283  ; 出料托框昇降Error detection
      OUT     L3220  ; 出料托框昇降異常
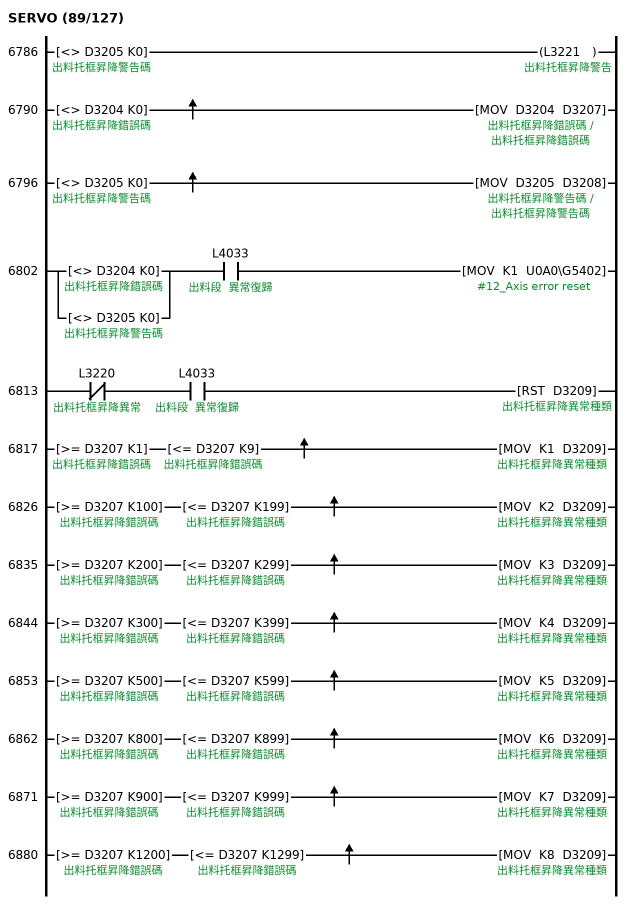
6786  LD<>    D3205 K0  ; 出料托框昇降警告碼
      OUT     L3221  ; 出料托框昇降警告
6790  LD<>    D3204 K0  ; 出料托框昇降錯誤碼
      MEP
      MOV     D3204 D3207  ; 出料托框昇降錯誤碼
6796  LD<>    D3205 K0  ; 出料托框昇降警告碼
      MEP
      MOV     D3205 D3208  ; 出料托框昇降警告碼
6802  LD<>    D3204 K0  ; 出料托框昇降錯誤碼
      OR<>    D3205 K0  ; 出料托框昇降警告碼
      AND     L4033  ; 出料段  異常復歸
      MOV     K1 U0A0\G5402  ; #12_Axis error reset
6813  LDI     L3220  ; 出料托框昇降異常
      AND     L4033  ; 出料段  異常復歸
      RST     D3209  ; 出料托框昇降異常種類
6817  LD>=    D3207 K1  ; 出料托框昇降錯誤碼
      AND<=   D3207 K9  ; 出料托框昇降錯誤碼
      MEP
      MOV     K1 D3209
6826  LD>=    D3207 K100  ; 出料托框昇降錯誤碼
      AND<=   D3207 K199  ; 出料托框昇降錯誤碼
      MEP
      MOV     K2 D3209
6835  LD>=    D3207 K200  ; 出料托框昇降錯誤碼
      AND<=   D3207 K299  ; 出料托框昇降錯誤碼
      MEP
      MOV     K3 D3209
6844  LD>=    D3207 K300  ; 出料托框昇降錯誤碼
      AND<=   D3207 K399  ; 出料托框昇降錯誤碼
      MEP
      MOV     K4 D3209
6853  LD>=    D3207 K500  ; 出料托框昇降錯誤碼
      AND<=   D3207 K599  ; 出料托框昇降錯誤碼
      MEP
      MOV     K5 D3209
6862  LD>=    D3207 K800  ; 出料托框昇降錯誤碼
      AND<=   D3207 K899  ; 出料托框昇降錯誤碼
      MEP
      MOV     K6 D3209
6871  LD>=    D3207 K900  ; 出料托框昇降錯誤碼
      AND<=   D3207 K999  ; 出料托框昇降錯誤碼
      MEP
      MOV     K7 D3209
6880  LD>=    D3207 K1200  ; 出料托框昇降錯誤碼
      AND<=   D3207 K1299  ; 出料托框昇降錯誤碼
      MEP
      MOV     K8 D3209
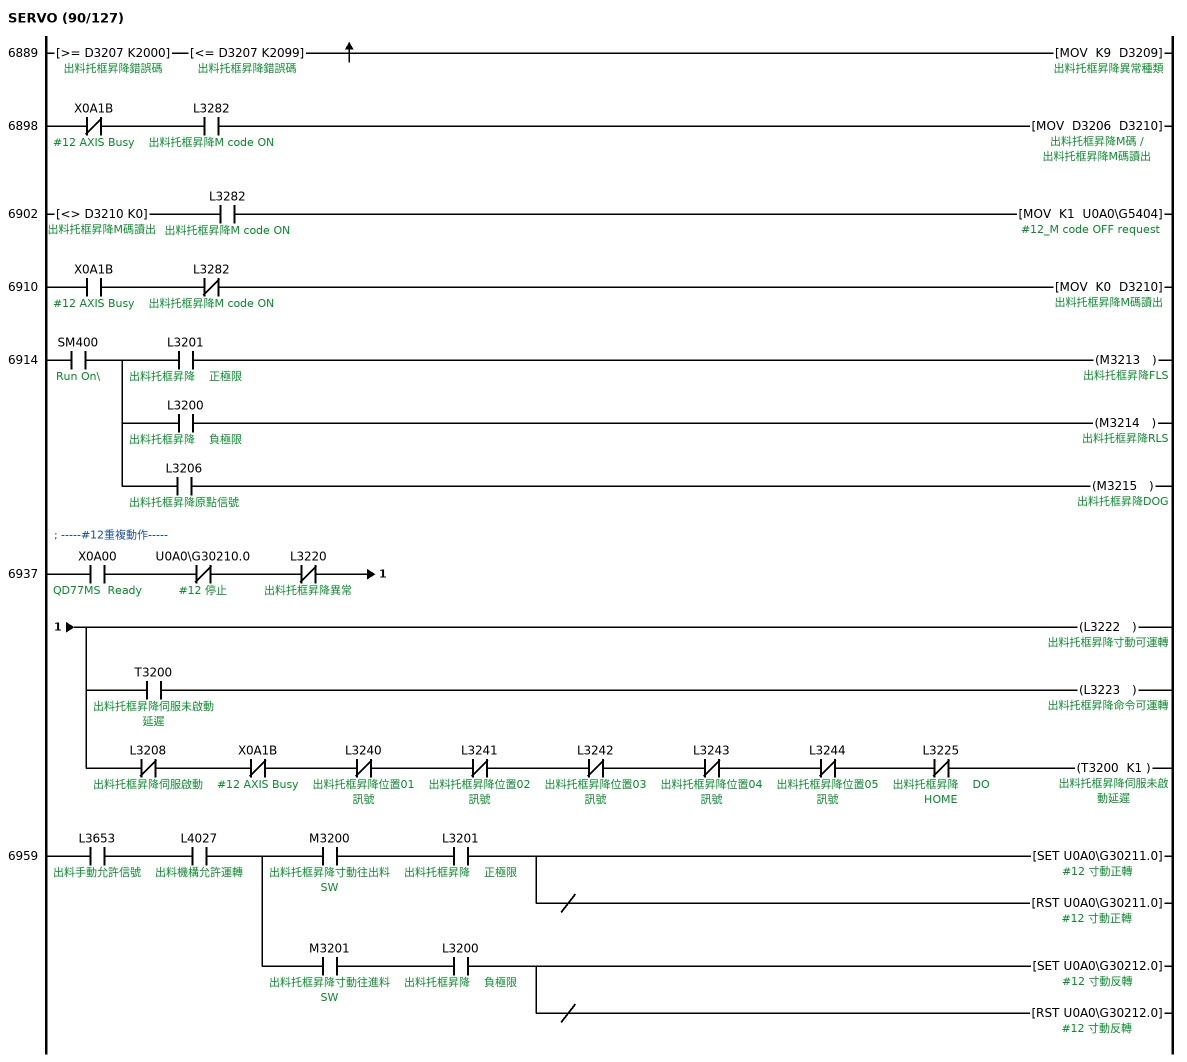
6889  LD>=    D3207 K2000  ; 出料托框昇降錯誤碼
      AND<=   D3207 K2099  ; 出料托框昇降錯誤碼
      MEP
      MOV     K9 D3209
6898  LDI     X0A1B  ; #12 AXIS Busy
      AND     L3282  ; 出料托框昇降M code ON
      MOV     D3206 D3210  ; 出料托框昇降M碼讀出
6902  LD<>    D3210 K0  ; 出料托框昇降M碼讀出
      AND     L3282  ; 出料托框昇降M code ON
      MOV     K1 U0A0\G5404  ; #12_M code OFF request
6910  LD      X0A1B  ; #12 AXIS Busy
      ANI     L3282  ; 出料托框昇降M code ON
      MOV     K0 D3210
6914  LD      SM400  ; Run On\
      MPS
      AND     L3201  ; 出料托框昇降    正極限
      OUT     M3213  ; 出料托框昇降FLS
      MRD
      AND     L3200  ; 出料托框昇降    負極限
      OUT     M3214  ; 出料托框昇降RLS
      MPP
      AND     L3206  ; 出料托框昇降原點信號
      OUT     M3215  ; 出料托框昇降DOG
; -----#12重複動作-----
6937  LD      X0A00  ; QD77MS  Ready
      ANI     U0A0\G30210.0  ; #12 停止
      ANI     L3220  ; 出料托框昇降異常
      OUT     L3222  ; 出料托框昇降寸動可運轉
      MPS
      AND     T3200  ; 出料托框昇降伺服未啟動延遲
      OUT     L3223  ; 出料托框昇降命令可運轉
      MPP
      ANI     L3208  ; 出料托框昇降伺服啟動
      ANI     X0A1B  ; #12 AXIS Busy
      ANI     L3240  ; 出料托框昇降位置01 訊號
      ANI     L3241  ; 出料托框昇降位置02 訊號
      ANI     L3242  ; 出料托框昇降位置03 訊號
      ANI     L3243  ; 出料托框昇降位置04 訊號
      ANI     L3244  ; 出料托框昇降位置05 訊號
      ANI     L3225  ; 出料托框昇降    DO HOME
      OUT     T3200 K1  ; 出料托框昇降伺服未啟動延遲
6959  LD      L3653  ; 出料手動允許信號
      AND     L4027  ; 出料機構允許運轉
      MPS
      AND     M3200  ; 出料托框昇降寸動往出料SW
      AND     L3201  ; 出料托框昇降    正極限
      SET     U0A0\G30211.0  ; #12 寸動正轉
      INV
      RST     U0A0\G30211.0  ; #12 寸動正轉
      MPP
      AND     M3201  ; 出料托框昇降寸動往進料SW
      AND     L3200  ; 出料托框昇降    負極限
      SET     U0A0\G30212.0  ; #12 寸動反轉
      INV
      RST     U0A0\G30212.0  ; #12 寸動反轉
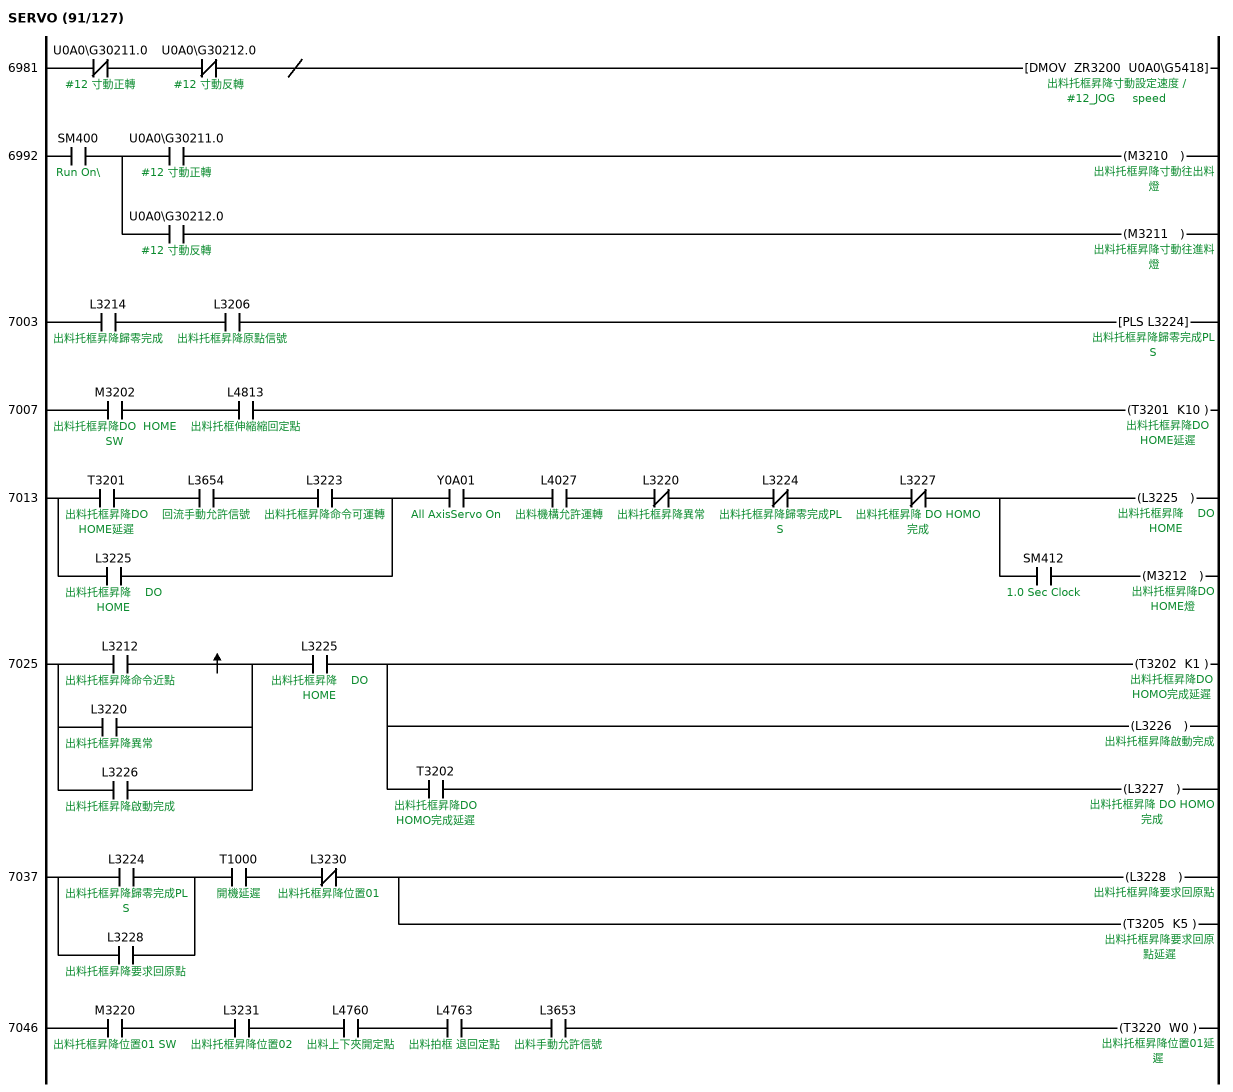
6981  LDI     U0A0\G30211.0  ; #12 寸動正轉
      ANI     U0A0\G30212.0  ; #12 寸動反轉
      INV
      DMOV    ZR3200 U0A0\G5418  ; 出料托框昇降寸動設定速度 / #12_JOG     speed
6992  LD      SM400  ; Run On\
      MPS
      AND     U0A0\G30211.0  ; #12 寸動正轉
      OUT     M3210  ; 出料托框昇降寸動往出料燈
      MPP
      AND     U0A0\G30212.0  ; #12 寸動反轉
      OUT     M3211  ; 出料托框昇降寸動往進料燈
7003  LD      L3214  ; 出料托框昇降歸零完成
      AND     L3206  ; 出料托框昇降原點信號
      PLS     L3224  ; 出料托框昇降歸零完成PLS
7007  LD      M3202  ; 出料托框昇降DO  HOME SW
      AND     L4813  ; 出料托框伸縮縮回定點
      OUT     T3201 K10  ; 出料托框昇降DO HOME延遲
7013  LD      T3201  ; 出料托框昇降DO HOME延遲
      AND     L3654  ; 回流手動允許信號
      AND     L3223  ; 出料托框昇降命令可運轉
      OR      L3225  ; 出料托框昇降    DO HOME
      AND     Y0A01  ; All AxisServo On
      AND     L4027  ; 出料機構允許運轉
      ANI     L3220  ; 出料托框昇降異常
      ANI     L3224  ; 出料托框昇降歸零完成PLS
      ANI     L3227  ; 出料托框昇降 DO HOMO 完成
      OUT     L3225  ; 出料托框昇降    DO HOME
      AND     SM412  ; 1.0 Sec Clock
      OUT     M3212  ; 出料托框昇降DO  HOME燈
7025  LD      L3212  ; 出料托框昇降命令近點
      MEP
      OR      L3220  ; 出料托框昇降異常
      OR      L3226  ; 出料托框昇降啟動完成
      AND     L3225  ; 出料托框昇降    DO HOME
      OUT     T3202 K1  ; 出料托框昇降DO HOMO完成延遲
      OUT     L3226  ; 出料托框昇降啟動完成
      AND     T3202  ; 出料托框昇降DO HOMO完成延遲
      OUT     L3227  ; 出料托框昇降 DO HOMO 完成
7037  LD      L3224  ; 出料托框昇降歸零完成PLS
      OR      L3228  ; 出料托框昇降要求回原點
      AND     T1000  ; 開機延遲
      ANI     L3230  ; 出料托框昇降位置01
      OUT     L3228  ; 出料托框昇降要求回原點
      OUT     T3205 K5  ; 出料托框昇降要求回原點延遲
7046  LD      M3220  ; 出料托框昇降位置01 SW
      AND     L3231  ; 出料托框昇降位置02
      AND     L4760  ; 出料上下夾開定點
      AND     L4763  ; 出料拍框 退回定點
      AND     L3653  ; 出料手動允許信號
      OUT     T3220 W0  ; 出料托框昇降位置01延遲
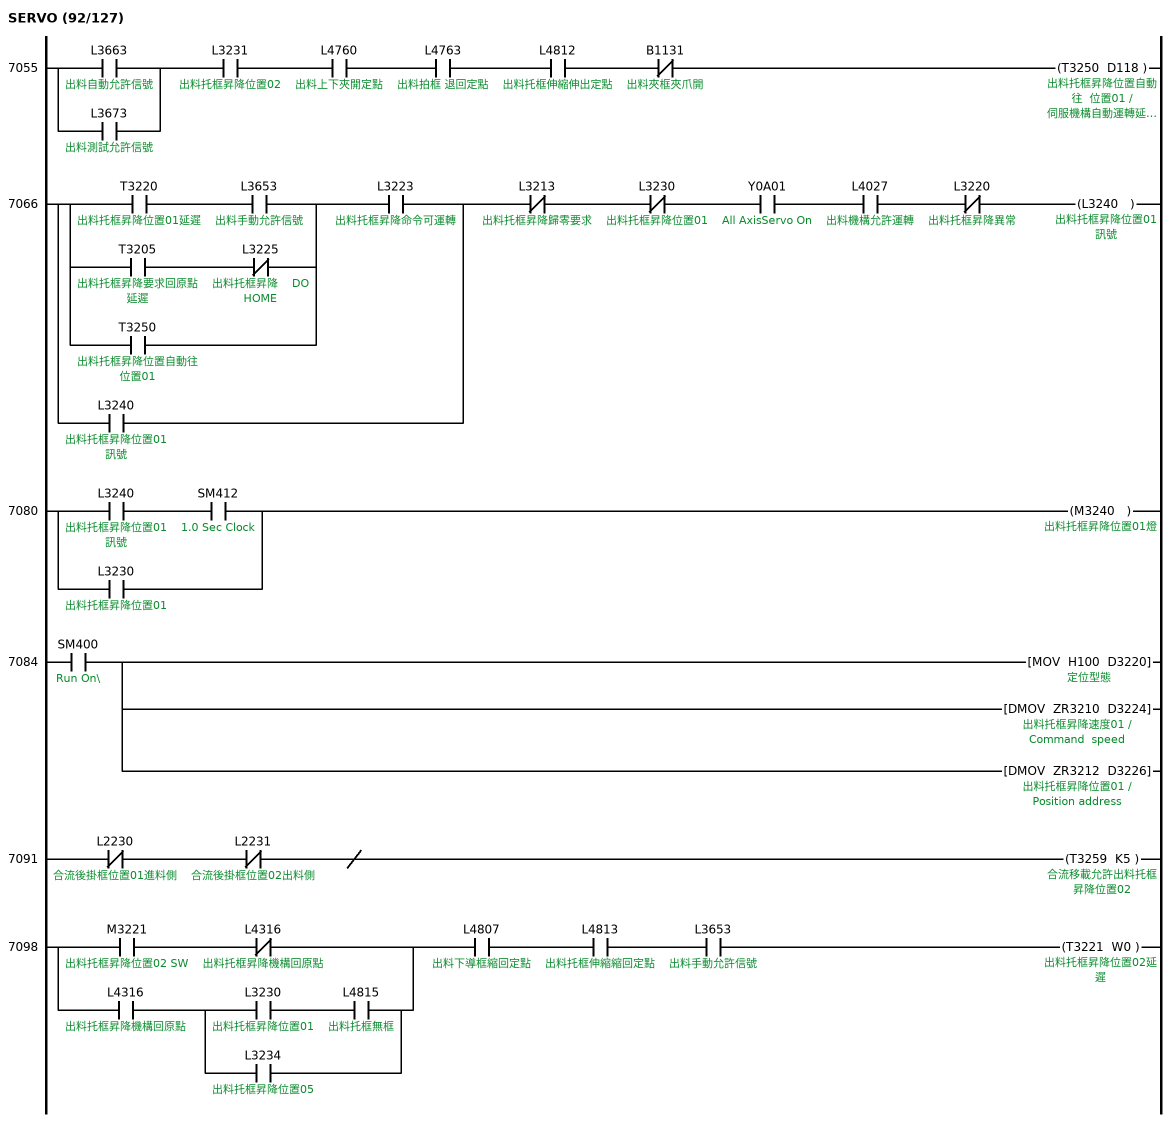
7055  LD      L3663  ; 出料自動允許信號
      OR      L3673  ; 出料測試允許信號
      AND     L3231  ; 出料托框昇降位置02
      AND     L4760  ; 出料上下夾開定點
      AND     L4763  ; 出料拍框 退回定點
      AND     L4812  ; 出料托框伸縮伸出定點
      ANI     B1131  ; 出料夾框夾爪開
      OUT     T3250 D118  ; 出料托框昇降位置自動往  位置01 / 伺服機構自動運轉延遲時間
7066  LD      T3220  ; 出料托框昇降位置01延遲
      AND     L3653  ; 出料手動允許信號
      LD      T3205  ; 出料托框昇降要求回原點延遲
      ANI     L3225  ; 出料托框昇降    DO HOME
      ORB
      OR      T3250  ; 出料托框昇降位置自動往  位置01
      AND     L3223  ; 出料托框昇降命令可運轉
      OR      L3240  ; 出料托框昇降位置01 訊號
      ANI     L3213  ; 出料托框昇降歸零要求
      ANI     L3230  ; 出料托框昇降位置01
      AND     Y0A01  ; All AxisServo On
      AND     L4027  ; 出料機構允許運轉
      ANI     L3220  ; 出料托框昇降異常
      OUT     L3240  ; 出料托框昇降位置01 訊號
7080  LD      L3240  ; 出料托框昇降位置01 訊號
      AND     SM412  ; 1.0 Sec Clock
      OR      L3230  ; 出料托框昇降位置01
      OUT     M3240  ; 出料托框昇降位置01燈
7084  LD      SM400  ; Run On\
      MOV     H100 D3220  ; 定位型態
      DMOV    ZR3210 D3224  ; 出料托框昇降速度01 / Command  speed
      DMOV    ZR3212 D3226  ; Position address
7091  LDI     L2230  ; 合流後掛框位置01進料側
      ANI     L2231  ; 合流後掛框位置02出料側
      INV
      OUT     T3259 K5  ; 合流移載允許出料托框昇降位置02
7098  LD      M3221  ; 出料托框昇降位置02 SW
      ANI     L4316  ; 出料托框昇降機構回原點
      LD      L4316  ; 出料托框昇降機構回原點
      LD      L3230  ; 出料托框昇降位置01
      AND     L4815  ; 出料托框無框
      OR      L3234  ; 出料托框昇降位置05
      ANB
      ORB
      AND     L4807  ; 出料下導框縮回定點
      AND     L4813  ; 出料托框伸縮縮回定點
      AND     L3653  ; 出料手動允許信號
      OUT     T3221 W0  ; 出料托框昇降位置02延遲
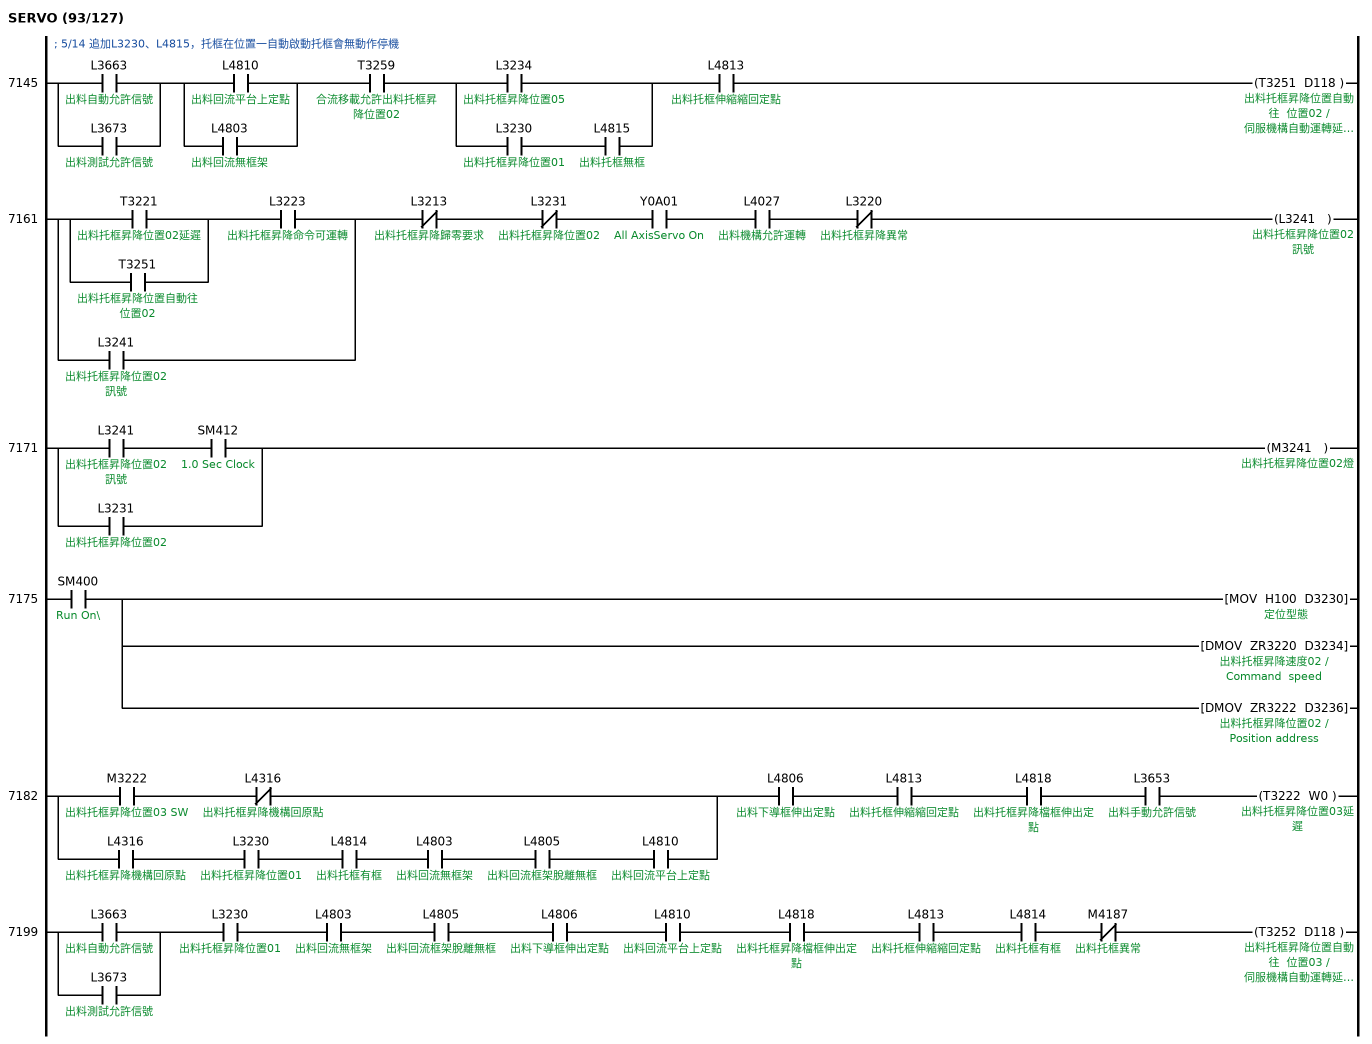
; 5/14 追加L3230、L4815，托框在位置一自動啟動托框會無動作停機
7145  LD      L3663  ; 出料自動允許信號
      OR      L3673  ; 出料測試允許信號
      LD      L4810  ; 出料回流平台上定點
      OR      L4803  ; 出料回流無框架
      ANB
      AND     T3259  ; 合流移載允許出料托框昇降位置02
      LD      L3234  ; 出料托框昇降位置05
      LD      L3230  ; 出料托框昇降位置01
      AND     L4815  ; 出料托框無框
      ORB
      ANB
      AND     L4813  ; 出料托框伸縮縮回定點
      OUT     T3251 D118  ; 出料托框昇降位置自動往  位置02 / 伺服機構自動運轉延遲時間
7161  LD      T3221  ; 出料托框昇降位置02延遲
      OR      T3251  ; 出料托框昇降位置自動往  位置02
      AND     L3223  ; 出料托框昇降命令可運轉
      OR      L3241  ; 出料托框昇降位置02 訊號
      ANI     L3213  ; 出料托框昇降歸零要求
      ANI     L3231  ; 出料托框昇降位置02
      AND     Y0A01  ; All AxisServo On
      AND     L4027  ; 出料機構允許運轉
      ANI     L3220  ; 出料托框昇降異常
      OUT     L3241  ; 出料托框昇降位置02 訊號
7171  LD      L3241  ; 出料托框昇降位置02 訊號
      AND     SM412  ; 1.0 Sec Clock
      OR      L3231  ; 出料托框昇降位置02
      OUT     M3241  ; 出料托框昇降位置02燈
7175  LD      SM400  ; Run On\
      MOV     H100 D3230  ; 定位型態
      DMOV    ZR3220 D3234  ; 出料托框昇降速度02 / Command  speed
      DMOV    ZR3222 D3236  ; Position address
7182  LD      M3222  ; 出料托框昇降位置03 SW
      ANI     L4316  ; 出料托框昇降機構回原點
      LD      L4316  ; 出料托框昇降機構回原點
      AND     L3230  ; 出料托框昇降位置01
      AND     L4814  ; 出料托框有框
      AND     L4803  ; 出料回流無框架
      AND     L4805  ; 出料回流框架脫離無框
      AND     L4810  ; 出料回流平台上定點
      ORB
      AND     L4806  ; 出料下導框伸出定點
      AND     L4813  ; 出料托框伸縮縮回定點
      AND     L4818  ; 出料托框昇降檔框伸出定點
      AND     L3653  ; 出料手動允許信號
      OUT     T3222 W0  ; 出料托框昇降位置03延遲
7199  LD      L3663  ; 出料自動允許信號
      OR      L3673  ; 出料測試允許信號
      AND     L3230  ; 出料托框昇降位置01
      AND     L4803  ; 出料回流無框架
      AND     L4805  ; 出料回流框架脫離無框
      AND     L4806  ; 出料下導框伸出定點
      AND     L4810  ; 出料回流平台上定點
      AND     L4818  ; 出料托框昇降檔框伸出定點
      AND     L4813  ; 出料托框伸縮縮回定點
      AND     L4814  ; 出料托框有框
      ANI     M4187  ; 出料托框異常
      OUT     T3252 D118  ; 出料托框昇降位置自動往  位置03 / 伺服機構自動運轉延遲時間
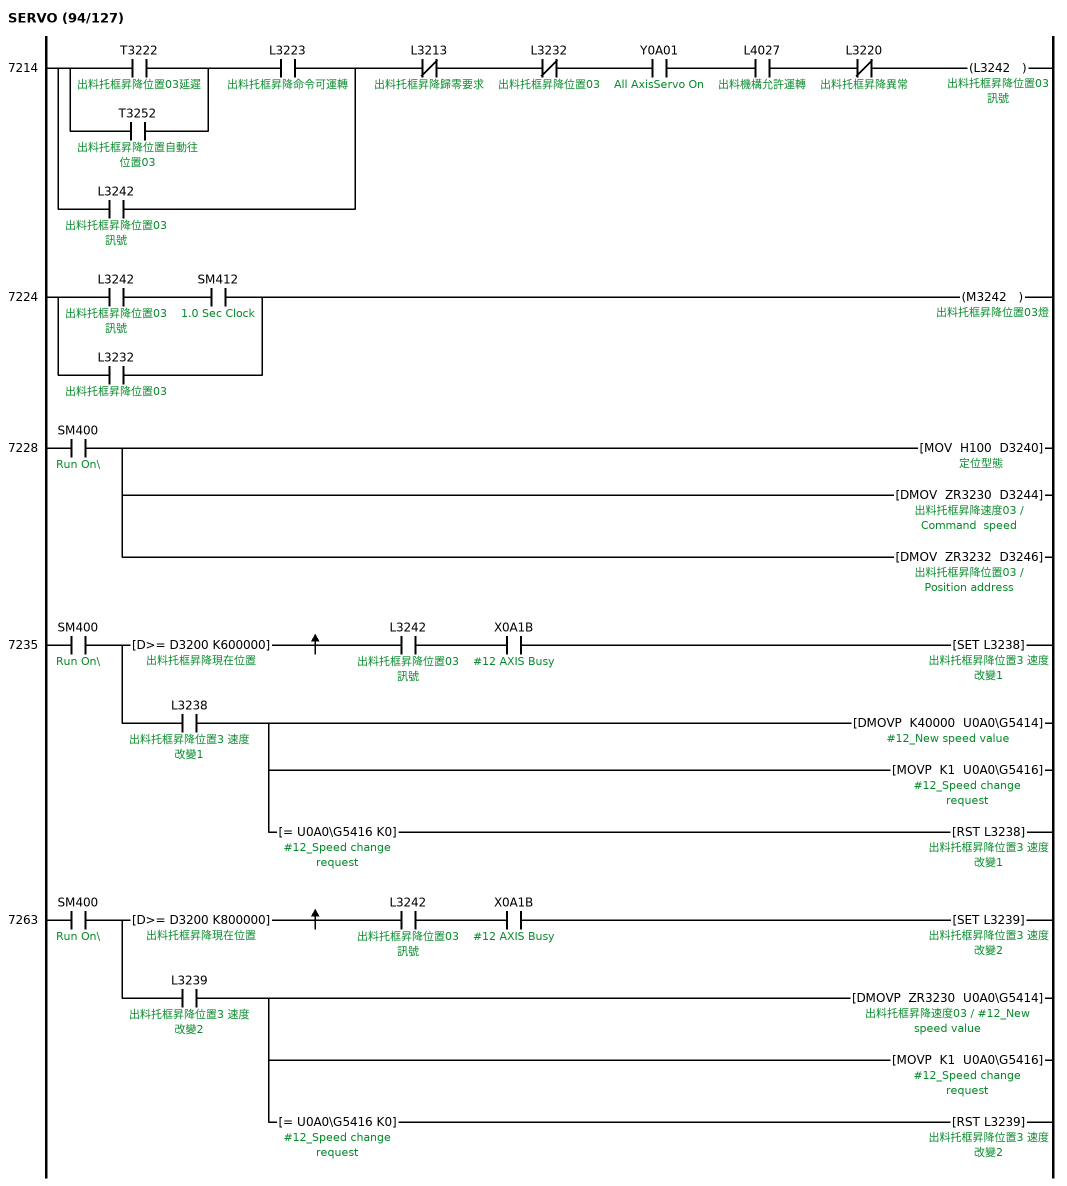
7214  LD      T3222  ; 出料托框昇降位置03延遲
      OR      T3252  ; 出料托框昇降位置自動往  位置03
      AND     L3223  ; 出料托框昇降命令可運轉
      OR      L3242  ; 出料托框昇降位置03 訊號
      ANI     L3213  ; 出料托框昇降歸零要求
      ANI     L3232  ; 出料托框昇降位置03
      AND     Y0A01  ; All AxisServo On
      AND     L4027  ; 出料機構允許運轉
      ANI     L3220  ; 出料托框昇降異常
      OUT     L3242  ; 出料托框昇降位置03 訊號
7224  LD      L3242  ; 出料托框昇降位置03 訊號
      AND     SM412  ; 1.0 Sec Clock
      OR      L3232  ; 出料托框昇降位置03
      OUT     M3242  ; 出料托框昇降位置03燈
7228  LD      SM400  ; Run On\
      MOV     H100 D3240  ; 定位型態
      DMOV    ZR3230 D3244  ; 出料托框昇降速度03 / Command  speed
      DMOV    ZR3232 D3246  ; Position address
7235  LD      SM400  ; Run On\
      MPS
      ANDD>=  D3200 K600000  ; 出料托框昇降現在位置
      MEP
      AND     L3242  ; 出料托框昇降位置03 訊號
      AND     X0A1B  ; #12 AXIS Busy
      SET     L3238  ; 出料托框昇降位置3 速度  改變1
      MPP
      AND     L3238  ; 出料托框昇降位置3 速度  改變1
      DMOVP   K40000 U0A0\G5414  ; #12_New speed value
      MOVP    K1 U0A0\G5416  ; #12_Speed change request
      AND=    U0A0\G5416 K0  ; #12_Speed change request
      RST     L3238  ; 出料托框昇降位置3 速度  改變1
7263  LD      SM400  ; Run On\
      MPS
      ANDD>=  D3200 K800000  ; 出料托框昇降現在位置
      MEP
      AND     L3242  ; 出料托框昇降位置03 訊號
      AND     X0A1B  ; #12 AXIS Busy
      SET     L3239  ; 出料托框昇降位置3 速度  改變2
      MPP
      AND     L3239  ; 出料托框昇降位置3 速度  改變2
      DMOVP   ZR3230 U0A0\G5414
      MOVP    K1 U0A0\G5416
      AND=    U0A0\G5416 K0  ; #12_Speed change request
      RST     L3239  ; 出料托框昇降位置3 速度  改變2
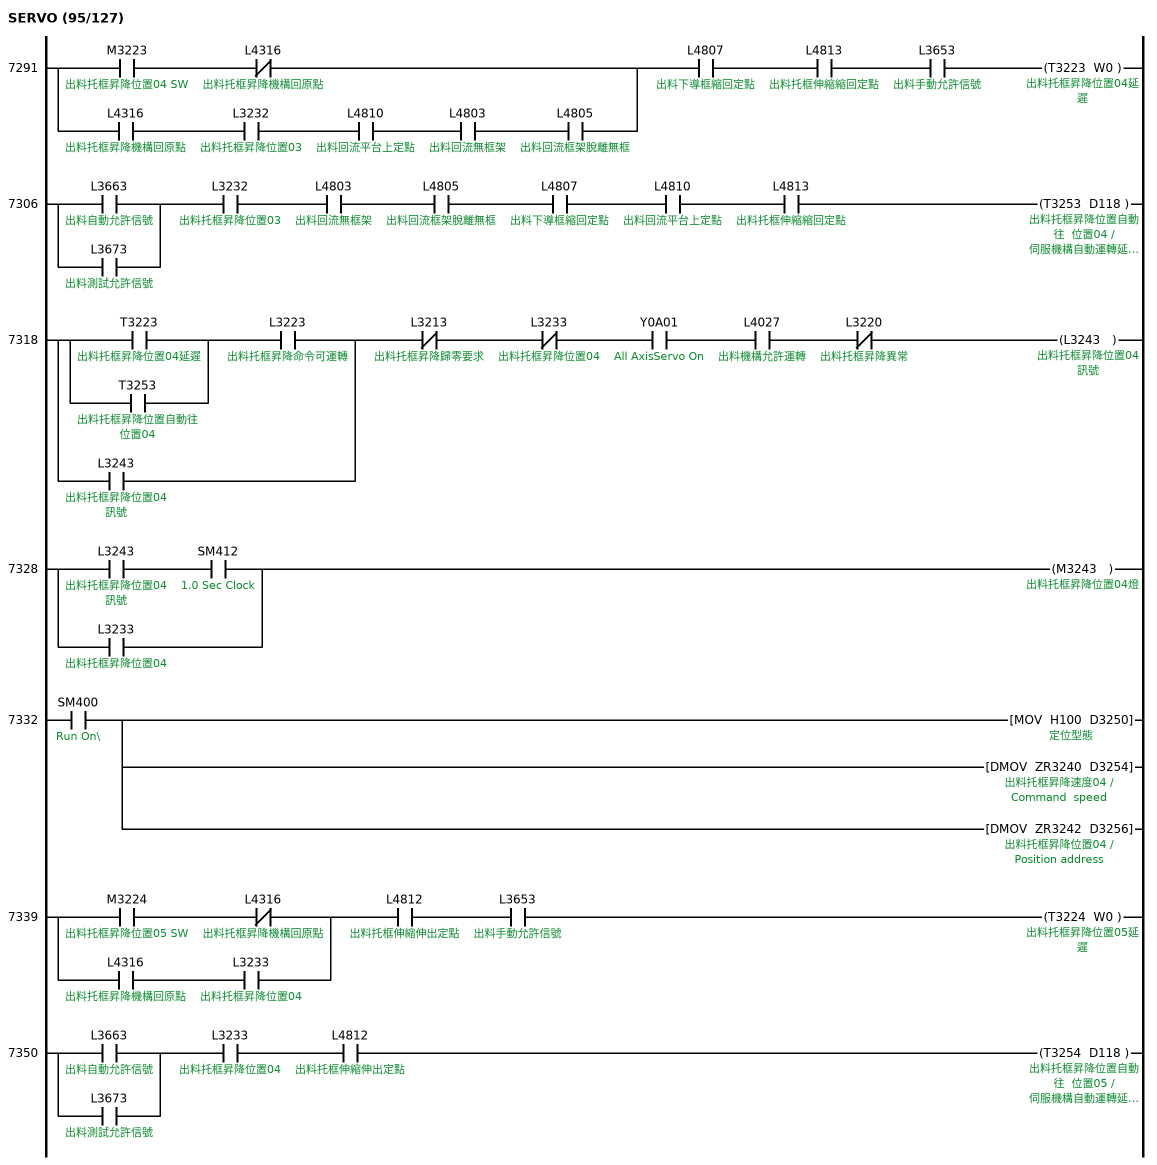
7291  LD      M3223  ; 出料托框昇降位置04 SW
      ANI     L4316  ; 出料托框昇降機構回原點
      LD      L4316  ; 出料托框昇降機構回原點
      AND     L3232  ; 出料托框昇降位置03
      AND     L4810  ; 出料回流平台上定點
      AND     L4803  ; 出料回流無框架
      AND     L4805  ; 出料回流框架脫離無框
      ORB
      AND     L4807  ; 出料下導框縮回定點
      AND     L4813  ; 出料托框伸縮縮回定點
      AND     L3653  ; 出料手動允許信號
      OUT     T3223 W0  ; 出料托框昇降位置04延遲
7306  LD      L3663  ; 出料自動允許信號
      OR      L3673  ; 出料測試允許信號
      AND     L3232  ; 出料托框昇降位置03
      AND     L4803  ; 出料回流無框架
      AND     L4805  ; 出料回流框架脫離無框
      AND     L4807  ; 出料下導框縮回定點
      AND     L4810  ; 出料回流平台上定點
      AND     L4813  ; 出料托框伸縮縮回定點
      OUT     T3253 D118  ; 出料托框昇降位置自動往  位置04 / 伺服機構自動運轉延遲時間
7318  LD      T3223  ; 出料托框昇降位置04延遲
      OR      T3253  ; 出料托框昇降位置自動往  位置04
      AND     L3223  ; 出料托框昇降命令可運轉
      OR      L3243  ; 出料托框昇降位置04 訊號
      ANI     L3213  ; 出料托框昇降歸零要求
      ANI     L3233  ; 出料托框昇降位置04
      AND     Y0A01  ; All AxisServo On
      AND     L4027  ; 出料機構允許運轉
      ANI     L3220  ; 出料托框昇降異常
      OUT     L3243  ; 出料托框昇降位置04 訊號
7328  LD      L3243  ; 出料托框昇降位置04 訊號
      AND     SM412  ; 1.0 Sec Clock
      OR      L3233  ; 出料托框昇降位置04
      OUT     M3243  ; 出料托框昇降位置04燈
7332  LD      SM400  ; Run On\
      MOV     H100 D3250  ; 定位型態
      DMOV    ZR3240 D3254  ; 出料托框昇降速度04 / Command  speed
      DMOV    ZR3242 D3256  ; Position address
7339  LD      M3224  ; 出料托框昇降位置05 SW
      ANI     L4316  ; 出料托框昇降機構回原點
      LD      L4316  ; 出料托框昇降機構回原點
      AND     L3233  ; 出料托框昇降位置04
      ORB
      AND     L4812  ; 出料托框伸縮伸出定點
      AND     L3653  ; 出料手動允許信號
      OUT     T3224 W0  ; 出料托框昇降位置05延遲
7350  LD      L3663  ; 出料自動允許信號
      OR      L3673  ; 出料測試允許信號
      AND     L3233  ; 出料托框昇降位置04
      AND     L4812  ; 出料托框伸縮伸出定點
      OUT     T3254 D118  ; 出料托框昇降位置自動往  位置05 / 伺服機構自動運轉延遲時間
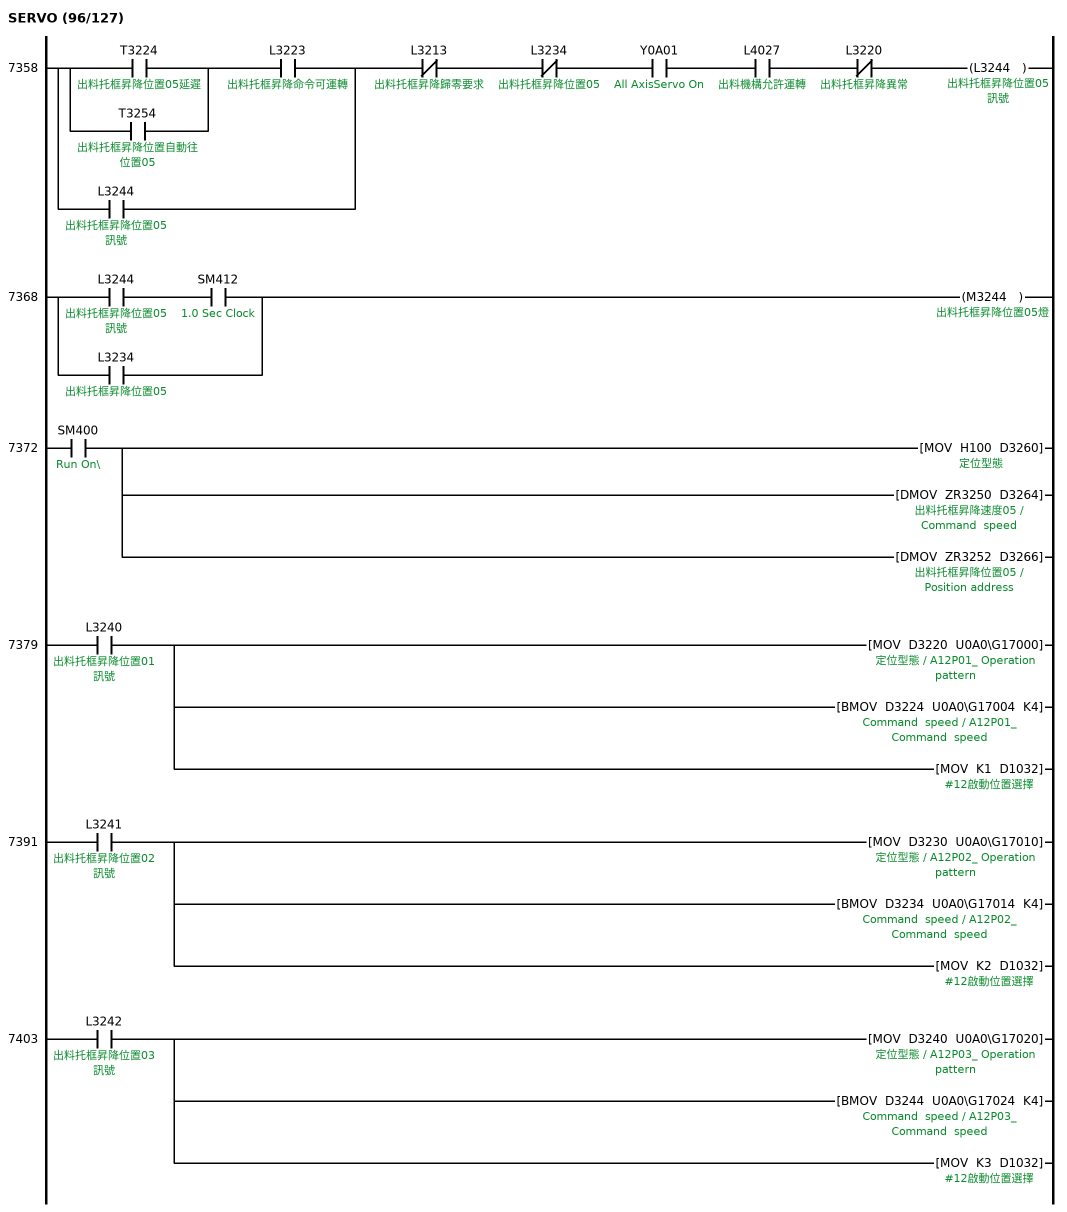
7358  LD      T3224  ; 出料托框昇降位置05延遲
      OR      T3254  ; 出料托框昇降位置自動往  位置05
      AND     L3223  ; 出料托框昇降命令可運轉
      OR      L3244  ; 出料托框昇降位置05 訊號
      ANI     L3213  ; 出料托框昇降歸零要求
      ANI     L3234  ; 出料托框昇降位置05
      AND     Y0A01  ; All AxisServo On
      AND     L4027  ; 出料機構允許運轉
      ANI     L3220  ; 出料托框昇降異常
      OUT     L3244  ; 出料托框昇降位置05 訊號
7368  LD      L3244  ; 出料托框昇降位置05 訊號
      AND     SM412  ; 1.0 Sec Clock
      OR      L3234  ; 出料托框昇降位置05
      OUT     M3244  ; 出料托框昇降位置05燈
7372  LD      SM400  ; Run On\
      MOV     H100 D3260  ; 定位型態
      DMOV    ZR3250 D3264  ; 出料托框昇降速度05 / Command  speed
      DMOV    ZR3252 D3266  ; Position address
7379  LD      L3240  ; 出料托框昇降位置01 訊號
      MOV     D3220 U0A0\G17000  ; A12P01_ Operation pattern
      BMOV    D3224 U0A0\G17004 K4  ; A12P01_ Command  speed
      MOV     K1 D1032  ; #12啟動位置選擇
7391  LD      L3241  ; 出料托框昇降位置02 訊號
      MOV     D3230 U0A0\G17010  ; A12P02_ Operation pattern
      BMOV    D3234 U0A0\G17014 K4  ; A12P02_ Command  speed
      MOV     K2 D1032
7403  LD      L3242  ; 出料托框昇降位置03 訊號
      MOV     D3240 U0A0\G17020  ; A12P03_ Operation pattern
      BMOV    D3244 U0A0\G17024 K4  ; A12P03_ Command  speed
      MOV     K3 D1032
